LIN {X 0,Y 430.337,Z 1009.214,A -85,B 0,C 180,E1 10047.011,E2 10047.011} C_VEL
LIN {X 0,Y 422.721,Z 1027.569,A -85,B 0,C 180,E1 10045.411,E2 10045.411} C_VEL
LIN {X 0,Y 412.935,Z 1049.67,A -85,B 0,C 180,E1 10043.164,E2 10043.164} C_VEL
LIN {X 0,Y 403.725,Z 1069.015,A -85,B 0,C 180,E1 10040.822,E2 10040.822} C_VEL
LIN {X 0,Y 396.125,Z 1084.43,A -85,B 0,C 180,E1 10038.672,E2 10038.672} C_VEL
LIN {X 0,Y 389.035,Z 1098.425,A -85,B 0,C 180,E1 10036.451,E2 10036.451} C_VEL
LIN {X 0,Y 381.874,Z 1112.344,A -85,B 0,C 180,E1 10033.937,E2 10033.937} C_VEL
LIN {X 0,Y 373.58,Z 1128.48,A -85,B 0,C 180,E1 10030.571,E2 10030.571} C_VEL
LIN {X 0,Y 366.042,Z 1142.999,A -85,B 0,C 180,E1 10026.939,E2 10026.939} C_VEL
LIN {X 0,Y 360.784,Z 1153.631,A -85,B 0,C 180,E1 10023.853,E2 10023.853} C_VEL
LIN {X 0,Y 356.104,Z 1163.538,A -85,B 0,C 180,E1 10020.546,E2 10020.546} C_VEL
LIN {X 0,Y 351.983,Z 1173.044,A -85,B 0,C 180,E1 10016.851,E2 10016.851} C_VEL
LIN {X 0,Y 348.273,Z 1182.759,A -85,B 0,C 180,E1 10012.27,E2 10012.27} C_VEL
LIN {X 0,Y 346.233,Z 1189.194,A -85,B 0,C 180,E1 10008.522,E2 10008.522} C_VEL
LIN {X 0,Y 345,Z 1194.199,A -85,B 0,C 180,E1 10004.948,E2 10004.948} C_VEL
LIN {X 0,Y 344.316,Z 1197.956,A -85,B 0,C 180,E1 10001.559,E2 10001.559} C_VEL
LIN {X 0,Y 344.025,Z 1200.753,A -85,B 0,C 180,E1 9998.188,E2 9998.188} C_VEL
LIN {X 0,Y 343.928,Z 1202.539,A -85,B 0,C 180,E1 9995.004,E2 9995.004} C_VEL
LIN {X 0,Y 343.912,Z 1203.491,A -85,B 0,C 180,E1 9991.833,E2 9991.833} C_VEL
LIN {X 0,Y 343.916,Z 1203.616,A -85,B 0,C 180,E1 9988.668,E2 9988.668} C_VEL
LIN {X 0,Y 343.921,Z 1202.851,A -85,B 0,C 180,E1 9985.331,E2 9985.331} C_VEL
LIN {X 0,Y 344.027,Z 1201.059,A -85,B 0,C 180,E1 9981.813,E2 9981.813} C_VEL
LIN {X 0,Y 344.324,Z 1198.421,A -85,B 0,C 180,E1 9978.442,E2 9978.442} C_VEL
LIN {X 0,Y 345.068,Z 1194.647,A -85,B 0,C 180,E1 9974.884,E2 9974.884} C_VEL
LIN {X 0,Y 346.354,Z 1189.832,A -85,B 0,C 180,E1 9971.311,E2 9971.311} C_VEL
LIN {X 0,Y 348.358,Z 1183.946,A -85,B 0,C 180,E1 9967.737,E2 9967.737} C_VEL
LIN {X 0,Y 351.492,Z 1176.249,A -85,B 0,C 180,E1 9963.838,E2 9963.838} C_VEL
LIN {X 0,Y 356.789,Z 1164.942,A -85,B 0,C 180,E1 9959.147,E2 9959.147} C_VEL
LIN {X 0,Y 362.173,Z 1154.455,A -85,B 0,C 180,E1 9955.532,E2 9955.532} C_VEL
LIN {X 0,Y 368.045,Z 1143.651,A -85,B 0,C 180,E1 9952.32,E2 9952.32} C_VEL
LIN {X 0,Y 375.262,Z 1130.896,A -85,B 0,C 180,E1 9949.046,E2 9949.046} C_VEL
LIN {X 0,Y 385.141,Z 1113.513,A -85,B 0,C 180,E1 9945.288,E2 9945.288} C_VEL
LIN {X 0,Y 393.592,Z 1098.51,A -85,B 0,C 180,E1 9942.549,E2 9942.549} C_VEL
LIN {X 0,Y 401.844,Z 1083.635,A -85,B 0,C 180,E1 9940.193,E2 9940.193} C_VEL
LIN {X 0,Y 410.984,Z 1066.687,A -85,B 0,C 180,E1 9937.865,E2 9937.865} C_VEL
LIN {X 0,Y 422.46,Z 1044.207,A -85,B 0,C 180,E1 9935.261,E2 9935.261} C_VEL
LIN {X 0,Y 431.379,Z 1025.581,A -85,B 0,C 180,E1 9933.445,E2 9933.445} C_VEL
LIN {X 0,Y 439.453,Z 1007.671,A -85,B 0,C 180,E1 9931.933,E2 9931.933} C_VEL
LIN {X 0,Y 447.149,Z 989.316,A -85,B 0,C 180,E1 9930.583,E2 9930.583} C_VEL
LIN {X 0,Y 456.108,Z 966.119,A -85,B 0,C 180,E1 9929.122,E2 9929.122} C_VEL
LIN {X 0,Y 464.642,Z 940.864,A -85,B 0,C 180,E1 9927.818,E2 9927.818} C_VEL
LIN {X 0,Y 470.596,Z 921.068,A -85,B 0,C 180,E1 9926.963,E2 9926.963} C_VEL
LIN {X 0,Y 476.118,Z 900.238,A -85,B 0,C 180,E1 9926.202,E2 9926.202} C_VEL
LIN {X 0,Y 481.006,Z 878.867,A -85,B 0,C 180,E1 9925.557,E2 9925.557} C_VEL
LIN {X 0,Y 485.675,Z 854.323,A -85,B 0,C 180,E1 9924.964,E2 9924.964} C_VEL
LIN {X 0,Y 489.575,Z 825.773,A -85,B 0,C 180,E1 9924.432,E2 9924.432} C_VEL
LIN {X 0,Y 495.874,Z 750.481,A -85,B 0,C 180,E1 9923.248,E2 9923.248} C_VEL
LIN {X 0,Y 512.566,Z 549.481,A -85,B 0,C 180,E1 9920.146,E2 9920.146} C_VEL
LIN {X 0,Y 508.739,Z 542.747,A -85,B 0,C 180,E1 9918.388,E2 9918.388} C_VEL
LIN {X 0,Y 504.17,Z 535.587,A -85,B 0,C 180,E1 9916.002,E2 9916.002} C_VEL
LIN {X 0,Y 501.343,Z 531.216,A -85,B 0,C 180,E1 9914.259,E2 9914.259} C_VEL
LIN {X 0,Y 498.781,Z 527.221,A -85,B 0,C 180,E1 9912.386,E2 9912.386} C_VEL
LIN {X 0,Y 496.043,Z 522.871,A -85,B 0,C 180,E1 9909.807,E2 9909.807} C_VEL
LIN {X 0,Y 493.101,Z 516.967,A -85,B 0,C 180,E1 9903.022,E2 9903.022} C_VEL
LIN {X 0,Y 493.133,Z 517.942,A -85,B 0,C 180,E1 9901.51,E2 9901.51} C_VEL
LIN {X 0,Y 495.468,Z 522.125,A -85,B 0,C 180,E1 9896.645,E2 9896.645} C_VEL
LIN {X 0,Y 496.115,Z 523.083,A -85,B 0,C 180,E1 9895.897,E2 9895.897} C_VEL
LIN {X 0,Y 499.395,Z 528.172,A -85,B 0,C 180,E1 9892.927,E2 9892.927} C_VEL
LIN {X 0,Y 502.886,Z 533.499,A -85,B 0,C 180,E1 9890.559,E2 9890.559} C_VEL
LIN {X 0,Y 506.125,Z 538.595,A -85,B 0,C 180,E1 9888.721,E2 9888.721} C_VEL
LIN {X 0,Y 510.891,Z 546.035,A -85,B 0,C 180,E1 9886.417,E2 9886.417} C_VEL
LIN {X 0,Y 512.516,Z 548.924,A -85,B 0,C 180,E1 9885.693,E2 9885.693} C_VEL
LIN {X 0,Y 495.201,Z 757.347,A -85,B 0,C 180,E1 9882.478,E2 9882.478} C_VEL
LIN {X 0,Y 489.709,Z 822.286,A -85,B 0,C 180,E1 9881.456,E2 9881.456} C_VEL
LIN {X 0,Y 485.517,Z 852.232,A -85,B 0,C 180,E1 9880.882,E2 9880.882} C_VEL
LIN {X 0,Y 481.117,Z 875.351,A -85,B 0,C 180,E1 9880.303,E2 9880.303} C_VEL
LIN {X 0,Y 476.393,Z 896.103,A -85,B 0,C 180,E1 9879.66,E2 9879.66} C_VEL
LIN {X 0,Y 471.007,Z 916.496,A -85,B 0,C 180,E1 9878.904,E2 9878.904} C_VEL
LIN {X 0,Y 464.448,Z 938.347,A -85,B 0,C 180,E1 9877.939,E2 9877.939} C_VEL
LIN {X 0,Y 455.544,Z 964.201,A -85,B 0,C 180,E1 9876.558,E2 9876.558} C_VEL
LIN {X 0,Y 447.584,Z 984.742,A -85,B 0,C 180,E1 9875.242,E2 9875.242} C_VEL
LIN {X 0,Y 439.887,Z 1003.084,A -85,B 0,C 180,E1 9873.875,E2 9873.875} C_VEL
LIN {X 0,Y 432.098,Z 1020.324,A -85,B 0,C 180,E1 9872.406,E2 9872.406} C_VEL
LIN {X 0,Y 423.37,Z 1038.473,A -85,B 0,C 180,E1 9870.628,E2 9870.628} C_VEL
LIN {X 0,Y 412.195,Z 1060.31,A -85,B 0,C 180,E1 9868.102,E2 9868.102} C_VEL
LIN {X 0,Y 402.856,Z 1077.491,A -85,B 0,C 180,E1 9865.739,E2 9865.739} C_VEL
LIN {X 0,Y 394.672,Z 1092.083,A -85,B 0,C 180,E1 9863.426,E2 9863.426} C_VEL
LIN {X 0,Y 386.658,Z 1106.09,A -85,B 0,C 180,E1 9860.875,E2 9860.875} C_VEL
LIN {X 0,Y 377.588,Z 1121.928,A -85,B 0,C 180,E1 9857.525,E2 9857.525} C_VEL
LIN {X 0,Y 369.258,Z 1136.254,A -85,B 0,C 180,E1 9853.883,E2 9853.883} C_VEL
LIN {X 0,Y 363.271,Z 1146.929,A -85,B 0,C 180,E1 9850.716,E2 9850.716} C_VEL
LIN {X 0,Y 358.211,Z 1156.378,A -85,B 0,C 180,E1 9847.481,E2 9847.481} C_VEL
LIN {X 0,Y 353.653,Z 1165.506,A -85,B 0,C 180,E1 9843.846,E2 9843.846} C_VEL
LIN {X 0,Y 349.353,Z 1175.205,A -85,B 0,C 180,E1 9839.196,E2 9839.196} C_VEL
LIN {X 0,Y 346.772,Z 1182.05,A -85,B 0,C 180,E1 9835.078,E2 9835.078} C_VEL
LIN {X 0,Y 345.352,Z 1186.792,A -85,B 0,C 180,E1 9831.573,E2 9831.573} C_VEL
LIN {X 0,Y 344.516,Z 1190.531,A -85,B 0,C 180,E1 9828.091,E2 9828.091} C_VEL
LIN {X 0,Y 344.106,Z 1193.313,A -85,B 0,C 180,E1 9824.619,E2 9824.619} C_VEL
LIN {X 0,Y 343.953,Z 1195.053,A -85,B 0,C 180,E1 9821.4,E2 9821.4} C_VEL
LIN {X 0,Y 343.924,Z 1195.977,A -85,B 0,C 180,E1 9818.189,E2 9818.189} C_VEL
LIN {X 0,Y 343.906,Z 1196.085,A -85,B 0,C 180,E1 9815.003,E2 9815.003} C_VEL
LIN {X 0,Y 343.931,Z 1195.318,A -85,B 0,C 180,E1 9811.665,E2 9811.665} C_VEL
LIN {X 0,Y 344.029,Z 1193.662,A -85,B 0,C 180,E1 9808.334,E2 9808.334} C_VEL
LIN {X 0,Y 344.331,Z 1190.956,A -85,B 0,C 180,E1 9804.835,E2 9804.835} C_VEL
LIN {X 0,Y 345.031,Z 1187.255,A -85,B 0,C 180,E1 9801.332,E2 9801.332} C_VEL
LIN {X 0,Y 346.236,Z 1182.539,A -85,B 0,C 180,E1 9797.829,E2 9797.829} C_VEL
LIN {X 0,Y 348.088,Z 1176.778,A -85,B 0,C 180,E1 9794.334,E2 9794.334} C_VEL
LIN {X 0,Y 350.975,Z 1169.245,A -85,B 0,C 180,E1 9790.529,E2 9790.529} C_VEL
LIN {X 0,Y 355.826,Z 1158.156,A -85,B 0,C 180,E1 9785.955,E2 9785.955} C_VEL
LIN {X 0,Y 360.768,Z 1147.87,A -85,B 0,C 180,E1 9782.429,E2 9782.429} C_VEL
LIN {X 0,Y 366.116,Z 1137.271,A -85,B 0,C 180,E1 9779.289,E2 9779.289} C_VEL
LIN {X 0,Y 372.644,Z 1124.746,A -85,B 0,C 180,E1 9776.075,E2 9776.075} C_VEL
LIN {X 0,Y 375.605,Z 1119.162,A -85,B 0,C 180,E1 9774.794,E2 9774.794} C_VEL
LIN {X 0,Y 376.92,Z 1115.143,A -85,B 0,C 180,E1 9773.809,E2 9773.809} C_VEL
LIN {X 0,Y 377.577,Z 1105.226,A -85,B 0,C 180,E1 9771.149,E2 9771.149} C_VEL
LIN {X 0,Y 379.228,Z 1100.831,A -85,B 0,C 180,E1 9770.204,E2 9770.204} C_VEL
LIN {X 0,Y 389.048,Z 1082.432,A -85,B 0,C 180,E1 9767.072,E2 9767.072} C_VEL
LIN {X 0,Y 397.703,Z 1065.618,A -85,B 0,C 180,E1 9764.642,E2 9764.642} C_VEL
LIN {X 0,Y 405.643,Z 1049.578,A -85,B 0,C 180,E1 9762.626,E2 9762.626} C_VEL
LIN {X 0,Y 414.307,Z 1031.223,A -85,B 0,C 180,E1 9760.623,E2 9760.623} C_VEL
LIN {X 0,Y 424.867,Z 1007.083,A -85,B 0,C 180,E1 9758.401,E2 9758.401} C_VEL
LIN {X 0,Y 432.771,Z 987.358,A -85,B 0,C 180,E1 9756.87,E2 9756.87} C_VEL
LIN {X 0,Y 440.027,Z 967.758,A -85,B 0,C 180,E1 9755.562,E2 9755.562} C_VEL
LIN {X 0,Y 446.974,Z 947.041,A -85,B 0,C 180,E1 9754.365,E2 9754.365} C_VEL
LIN {X 0,Y 455.108,Z 919.496,A -85,B 0,C 180,E1 9753.053,E2 9753.053} C_VEL
LIN {X 0,Y 460.585,Z 897.814,A -85,B 0,C 180,E1 9752.209,E2 9752.209} C_VEL
LIN {X 0,Y 465.192,Z 876.616,A -85,B 0,C 180,E1 9751.522,E2 9751.522} C_VEL
LIN {X 0,Y 469.15,Z 854.894,A -85,B 0,C 180,E1 9750.948,E2 9750.948} C_VEL
LIN {X 0,Y 473.042,Z 827.866,A -85,B 0,C 180,E1 9750.39,E2 9750.39} C_VEL
LIN {X 0,Y 476.588,Z 784.854,A -85,B 0,C 180,E1 9749.693,E2 9749.693} C_VEL
LIN {X 0,Y 493.006,Z 566.419,A -85,B 0,C 180,E1 9746.295,E2 9746.295} C_VEL
LIN {X 0,Y 494.586,Z 545.42,A -85,B 0,C 180,E1 9745.957,E2 9745.957} C_VEL
LIN {X 0,Y 487.433,Z 533.892,A -85,B 0,C 180,E1 9743.355,E2 9743.355} C_VEL
LIN {X 0,Y 480.969,Z 523.893,A -85,B 0,C 180,E1 9740.633,E2 9740.633} C_VEL
LIN {X 0,Y 475.999,Z 516.443,A -85,B 0,C 180,E1 9738.176,E2 9738.176} C_VEL
LIN {X 0,Y 472.598,Z 511.532,A -85,B 0,C 180,E1 9736.217,E2 9736.217} C_VEL
LIN {X 0,Y 469.595,Z 507.098,A -85,B 0,C 180,E1 9734.174,E2 9734.174} C_VEL
LIN {X 0,Y 466.586,Z 502.594,A -85,B 0,C 180,E1 9731.621,E2 9731.621} C_VEL
LIN {X 0,Y 463.469,Z 498.329,A -85,B 0,C 180,E1 9727.687,E2 9727.687} C_VEL
LIN {X 0,Y 462.965,Z 496.787,A -85,B 0,C 180,E1 9726.448,E2 9726.448} C_VEL
LIN {X 0,Y 462.675,Z 496.688,A -85,B 0,C 180,E1 9720.371,E2 9720.371} C_VEL
LIN {X 0,Y 463.125,Z 497.115,A -85,B 0,C 180,E1 9719.258,E2 9719.258} C_VEL
LIN {X 0,Y 464.849,Z 500.839,A -85,B 0,C 180,E1 9716.3,E2 9716.3} C_VEL
LIN {X 0,Y 466.718,Z 502.888,A -85,B 0,C 180,E1 9714.344,E2 9714.344} C_VEL
LIN {X 0,Y 469.77,Z 507.346,A -85,B 0,C 180,E1 9711.801,E2 9711.801} C_VEL
LIN {X 0,Y 473.776,Z 513.252,A -85,B 0,C 180,E1 9709.174,E2 9709.174} C_VEL
LIN {X 0,Y 478.001,Z 519.572,A -85,B 0,C 180,E1 9706.882,E2 9706.882} C_VEL
LIN {X 0,Y 482.852,Z 526.838,A -85,B 0,C 180,E1 9704.629,E2 9704.629} C_VEL
LIN {X 0,Y 489.094,Z 536.563,A -85,B 0,C 180,E1 9702.111,E2 9702.111} C_VEL
LIN {X 0,Y 493.408,Z 544.162,A -85,B 0,C 180,E1 9700.527,E2 9700.527} C_VEL
LIN {X 0,Y 494.638,Z 546.737,A -85,B 0,C 180,E1 9700.084,E2 9700.084} C_VEL
LIN {X 0,Y 477.921,Z 768.344,A -85,B 0,C 180,E1 9696.639,E2 9696.639} C_VEL
LIN {X 0,Y 473.332,Z 827.257,A -85,B 0,C 180,E1 9695.7,E2 9695.7} C_VEL
LIN {X 0,Y 469.295,Z 857.376,A -85,B 0,C 180,E1 9695.108,E2 9695.108} C_VEL
LIN {X 0,Y 465.131,Z 880.202,A -85,B 0,C 180,E1 9694.528,E2 9694.528} C_VEL
LIN {X 0,Y 460.653,Z 900.854,A -85,B 0,C 180,E1 9693.878,E2 9693.878} C_VEL
LIN {X 0,Y 455.634,Z 920.879,A -85,B 0,C 180,E1 9693.123,E2 9693.123} C_VEL
LIN {X 0,Y 449.408,Z 942.77,A -85,B 0,C 180,E1 9692.145,E2 9692.145} C_VEL
LIN {X 0,Y 440.755,Z 969.366,A -85,B 0,C 180,E1 9690.702,E2 9690.702} C_VEL
LIN {X 0,Y 433.36,Z 989.619,A -85,B 0,C 180,E1 9689.386,E2 9689.386} C_VEL
LIN {X 0,Y 425.854,Z 1008.604,A -85,B 0,C 180,E1 9687.953,E2 9687.953} C_VEL
LIN {X 0,Y 418.291,Z 1026.382,A -85,B 0,C 180,E1 9686.414,E2 9686.414} C_VEL
LIN {X 0,Y 409.052,Z 1046.833,A -85,B 0,C 180,E1 9684.367,E2 9684.367} C_VEL
LIN {X 0,Y 398.982,Z 1067.537,A -85,B 0,C 180,E1 9681.898,E2 9681.898} C_VEL
LIN {X 0,Y 390.791,Z 1083.647,A -85,B 0,C 180,E1 9679.659,E2 9679.659} C_VEL
LIN {X 0,Y 383.252,Z 1098.048,A -85,B 0,C 180,E1 9677.368,E2 9677.368} C_VEL
LIN {X 0,Y 375.365,Z 1112.862,A -85,B 0,C 180,E1 9674.665,E2 9674.665} C_VEL
LIN {X 0,Y 366.459,Z 1129.485,A -85,B 0,C 180,E1 9671.115,E2 9671.115} C_VEL
LIN {X 0,Y 359.007,Z 1143.306,A -85,B 0,C 180,E1 9667.586,E2 9667.586} C_VEL
LIN {X 0,Y 353.534,Z 1153.902,A -85,B 0,C 180,E1 9664.448,E2 9664.448} C_VEL
LIN {X 0,Y 348.669,Z 1163.773,A -85,B 0,C 180,E1 9661.077,E2 9661.077} C_VEL
LIN {X 0,Y 343.854,Z 1174.5,A -85,B 0,C 180,E1 9656.782,E2 9656.782} C_VEL
LIN {X 0,Y 340.36,Z 1183.199,A -85,B 0,C 180,E1 9652.452,E2 9652.452} C_VEL
LIN {X 0,Y 338.336,Z 1189.291,A -85,B 0,C 180,E1 9648.792,E2 9648.792} C_VEL
LIN {X 0,Y 337.091,Z 1194.053,A -85,B 0,C 180,E1 9645.308,E2 9645.308} C_VEL
LIN {X 0,Y 336.353,Z 1197.825,A -85,B 0,C 180,E1 9641.837,E2 9641.837} C_VEL
LIN {X 0,Y 336.036,Z 1200.635,A -85,B 0,C 180,E1 9638.384,E2 9638.384} C_VEL
LIN {X 0,Y 335.93,Z 1202.433,A -85,B 0,C 180,E1 9635.124,E2 9635.124} C_VEL
LIN {X 0,Y 335.913,Z 1203.397,A -85,B 0,C 180,E1 9631.877,E2 9631.877} C_VEL
LIN {X 0,Y 335.916,Z 1203.535,A -85,B 0,C 180,E1 9628.636,E2 9628.636} C_VEL
LIN {X 0,Y 335.923,Z 1202.781,A -85,B 0,C 180,E1 9625.22,E2 9625.22} C_VEL
LIN {X 0,Y 336.036,Z 1201,A -85,B 0,C 180,E1 9621.617,E2 9621.617} C_VEL
LIN {X 0,Y 336.361,Z 1198.374,A -85,B 0,C 180,E1 9618.165,E2 9618.165} C_VEL
LIN {X 0,Y 337.166,Z 1194.615,A -85,B 0,C 180,E1 9614.521,E2 9614.521} C_VEL
LIN {X 0,Y 338.547,Z 1189.813,A -85,B 0,C 180,E1 9610.864,E2 9610.864} C_VEL
LIN {X 0,Y 340.694,Z 1183.943,A -85,B 0,C 180,E1 9607.208,E2 9607.208} C_VEL
LIN {X 0,Y 343.855,Z 1176.617,A -85,B 0,C 180,E1 9603.398,E2 9603.398} C_VEL
LIN {X 0,Y 349.172,Z 1165.906,A -85,B 0,C 180,E1 9598.782,E2 9598.782} C_VEL
LIN {X 0,Y 355.003,Z 1155.038,A -85,B 0,C 180,E1 9594.931,E2 9594.931} C_VEL
LIN {X 0,Y 361.115,Z 1144.315,A -85,B 0,C 180,E1 9591.668,E2 9591.668} C_VEL
LIN {X 0,Y 368.027,Z 1132.577,A -85,B 0,C 180,E1 9588.579,E2 9588.579} C_VEL
LIN {X 0,Y 377.097,Z 1117.416,A -85,B 0,C 180,E1 9585.147,E2 9585.147} C_VEL
LIN {X 0,Y 387.052,Z 1100.377,A -85,B 0,C 180,E1 9581.928,E2 9581.928} C_VEL
LIN {X 0,Y 396.019,Z 1084.777,A -85,B 0,C 180,E1 9579.414,E2 9579.414} C_VEL
LIN {X 0,Y 404.635,Z 1069.353,A -85,B 0,C 180,E1 9577.259,E2 9577.259} C_VEL
LIN {X 0,Y 413.667,Z 1052.517,A -85,B 0,C 180,E1 9575.218,E2 9575.218} C_VEL
LIN {X 0,Y 424.884,Z 1030.346,A -85,B 0,C 180,E1 9572.93,E2 9572.93} C_VEL
LIN {X 0,Y 434.172,Z 1010.429,A -85,B 0,C 180,E1 9571.21,E2 9571.21} C_VEL
LIN {X 0,Y 442.148,Z 992.041,A -85,B 0,C 180,E1 9569.836,E2 9569.836} C_VEL
LIN {X 0,Y 449.827,Z 972.877,A -85,B 0,C 180,E1 9568.599,E2 9568.599} C_VEL
LIN {X 0,Y 457.246,Z 952.607,A -85,B 0,C 180,E1 9567.478,E2 9567.478} C_VEL
LIN {X 0,Y 465.609,Z 926.935,A -85,B 0,C 180,E1 9566.291,E2 9566.291} C_VEL
LIN {X 0,Y 472.3,Z 902.65,A -85,B 0,C 180,E1 9565.387,E2 9565.387} C_VEL
LIN {X 0,Y 477.432,Z 880.973,A -85,B 0,C 180,E1 9564.726,E2 9564.726} C_VEL
LIN {X 0,Y 481.653,Z 859.76,A -85,B 0,C 180,E1 9564.203,E2 9564.203} C_VEL
LIN {X 0,Y 485.58,Z 834.829,A -85,B 0,C 180,E1 9563.709,E2 9563.709} C_VEL
LIN {X 0,Y 489.174,Z 798.01,A -85,B 0,C 180,E1 9563.109,E2 9563.109} C_VEL
LIN {X 0,Y 507.912,Z 575.83,A -85,B 0,C 180,E1 9559.692,E2 9559.692} C_VEL
LIN {X 0,Y 509.714,Z 554.831,A -85,B 0,C 180,E1 9559.361,E2 9559.361} C_VEL
LIN {X 0,Y 505.974,Z 548.265,A -85,B 0,C 180,E1 9557.54,E2 9557.54} C_VEL
LIN {X 0,Y 502.226,Z 542.441,A -85,B 0,C 180,E1 9555.473,E2 9555.473} C_VEL
LIN {X 0,Y 499.942,Z 538.803,A -85,B 0,C 180,E1 9554.005,E2 9554.005} C_VEL
LIN {X 0,Y 497.519,Z 534.955,A -85,B 0,C 180,E1 9552.182,E2 9552.182} C_VEL
LIN {X 0,Y 494.879,Z 530.602,A -85,B 0,C 180,E1 9549.61,E2 9549.61} C_VEL
LIN {X 0,Y 492.117,Z 525.419,A -85,B 0,C 180,E1 9543.728,E2 9543.728} C_VEL
LIN {X 0,Y 492.128,Z 524.917,A -85,B 0,C 180,E1 9542.678,E2 9542.678} C_VEL
LIN {X 0,Y 494.389,Z 530.008,A -85,B 0,C 180,E1 9536.754,E2 9536.754} C_VEL
LIN {X 0,Y 495.021,Z 530.988,A -85,B 0,C 180,E1 9536.004,E2 9536.004} C_VEL
LIN {X 0,Y 498.178,Z 535.986,A -85,B 0,C 180,E1 9533.083,E2 9533.083} C_VEL
LIN {X 0,Y 501.521,Z 541.18,A -85,B 0,C 180,E1 9530.764,E2 9530.764} C_VEL
LIN {X 0,Y 504.699,Z 546.29,A -85,B 0,C 180,E1 9528.92,E2 9528.92} C_VEL
LIN {X 0,Y 509.327,Z 553.688,A -85,B 0,C 180,E1 9526.634,E2 9526.634} C_VEL
LIN {X 0,Y 509.654,Z 554.618,A -85,B 0,C 180,E1 9526.467,E2 9526.467} C_VEL
LIN {X 0,Y 491.699,Z 765.89,A -85,B 0,C 180,E1 9523.22,E2 9523.22} C_VEL
LIN {X 0,Y 486.687,Z 823.199,A -85,B 0,C 180,E1 9522.319,E2 9522.319} C_VEL
LIN {X 0,Y 482.354,Z 853.133,A -85,B 0,C 180,E1 9521.745,E2 9521.745} C_VEL
LIN {X 0,Y 477.962,Z 875.7,A -85,B 0,C 180,E1 9521.184,E2 9521.184} C_VEL
LIN {X 0,Y 473.183,Z 896.258,A -85,B 0,C 180,E1 9520.553,E2 9520.553} C_VEL
LIN {X 0,Y 467.503,Z 917.296,A -85,B 0,C 180,E1 9519.779,E2 9519.779} C_VEL
LIN {X 0,Y 459.94,Z 941.852,A -85,B 0,C 180,E1 9518.69,E2 9518.69} C_VEL
LIN {X 0,Y 451.18,Z 966.167,A -85,B 0,C 180,E1 9517.37,E2 9517.37} C_VEL
LIN {X 0,Y 443.411,Z 985.678,A -85,B 0,C 180,E1 9516.117,E2 9516.117} C_VEL
LIN {X 0,Y 435.536,Z 1003.933,A -85,B 0,C 180,E1 9514.757,E2 9514.757} C_VEL
LIN {X 0,Y 427.233,Z 1021.787,A -85,B 0,C 180,E1 9513.231,E2 9513.231} C_VEL
LIN {X 0,Y 416.762,Z 1042.929,A -85,B 0,C 180,E1 9511.125,E2 9511.125} C_VEL
LIN {X 0,Y 405.951,Z 1062.989,A -85,B 0,C 180,E1 9508.723,E2 9508.723} C_VEL
LIN {X 0,Y 397.16,Z 1078.624,A -85,B 0,C 180,E1 9506.54,E2 9506.54} C_VEL
LIN {X 0,Y 388.54,Z 1093.452,A -85,B 0,C 180,E1 9504.156,E2 9504.156} C_VEL
LIN {X 0,Y 378.838,Z 1109.866,A -85,B 0,C 180,E1 9501.085,E2 9501.085} C_VEL
LIN {X 0,Y 369.067,Z 1125.951,A -85,B 0,C 180,E1 9497.467,E2 9497.467} C_VEL
LIN {X 0,Y 361.894,Z 1137.891,A -85,B 0,C 180,E1 9494.307,E2 9494.307} C_VEL
LIN {X 0,Y 355.798,Z 1148.309,A -85,B 0,C 180,E1 9491.116,E2 9491.116} C_VEL
LIN {X 0,Y 349.609,Z 1159.485,A -85,B 0,C 180,E1 9487.117,E2 9487.117} C_VEL
LIN {X 0,Y 344.198,Z 1170,A -85,B 0,C 180,E1 9482.507,E2 9482.507} C_VEL
LIN {X 0,Y 340.989,Z 1177.103,A -85,B 0,C 180,E1 9478.743,E2 9478.743} C_VEL
LIN {X 0,Y 338.743,Z 1182.956,A -85,B 0,C 180,E1 9475.015,E2 9475.015} C_VEL
LIN {X 0,Y 337.243,Z 1187.805,A -85,B 0,C 180,E1 9471.205,E2 9471.205} C_VEL
LIN {X 0,Y 336.353,Z 1191.972,A -85,B 0,C 180,E1 9466.937,E2 9466.937} C_VEL
LIN {X 0,Y 335.99,Z 1194.765,A -85,B 0,C 180,E1 9462.546,E2 9462.546} C_VEL
LIN {X 0,Y 335.925,Z 1196.009,A -85,B 0,C 180,E1 9458.731,E2 9458.731} C_VEL
LIN {X 0,Y 335.906,Z 1196.186,A -85,B 0,C 180,E1 9455.123,E2 9455.123} C_VEL
LIN {X 0,Y 335.931,Z 1195.444,A -85,B 0,C 180,E1 9451.705,E2 9451.705} C_VEL
LIN {X 0,Y 336.032,Z 1193.813,A -85,B 0,C 180,E1 9448.294,E2 9448.294} C_VEL
LIN {X 0,Y 336.348,Z 1191.134,A -85,B 0,C 180,E1 9444.712,E2 9444.712} C_VEL
LIN {X 0,Y 337.085,Z 1187.459,A -85,B 0,C 180,E1 9441.126,E2 9441.126} C_VEL
LIN {X 0,Y 338.363,Z 1182.768,A -85,B 0,C 180,E1 9437.542,E2 9437.542} C_VEL
LIN {X 0,Y 340.299,Z 1177.034,A -85,B 0,C 180,E1 9433.966,E2 9433.966} C_VEL
LIN {X 0,Y 343.03,Z 1170.217,A -85,B 0,C 180,E1 9430.414,E2 9430.414} C_VEL
LIN {X 0,Y 347.6,Z 1160.28,A -85,B 0,C 180,E1 9426.071,E2 9426.071} C_VEL
LIN {X 0,Y 353.312,Z 1148.738,A -85,B 0,C 180,E1 9421.979,E2 9421.979} C_VEL
LIN {X 0,Y 358.833,Z 1138.222,A -85,B 0,C 180,E1 9418.782,E2 9418.782} C_VEL
LIN {X 0,Y 365.224,Z 1126.409,A -85,B 0,C 180,E1 9415.669,E2 9415.669} C_VEL
LIN {X 0,Y 373.681,Z 1111.126,A -85,B 0,C 180,E1 9412.211,E2 9412.211} C_VEL
LIN {X 0,Y 379.228,Z 1100.831,A -85,B 0,C 180,E1 9410.204,E2 9410.204} C_VEL
LIN {X 0,Y 380.941,Z 1096.425,A -85,B 0,C 180,E1 9409.276,E2 9409.276} C_VEL
LIN {X 0,Y 382.709,Z 1084.847,A -85,B 0,C 180,E1 9406.621,E2 9406.621} C_VEL
LIN {X 0,Y 384.413,Z 1080.641,A -85,B 0,C 180,E1 9405.89,E2 9405.89} C_VEL
LIN {X 0,Y 392.59,Z 1065.226,A -85,B 0,C 180,E1 9403.671,E2 9403.671} C_VEL
LIN {X 0,Y 400.776,Z 1049.133,A -85,B 0,C 180,E1 9401.65,E2 9401.65} C_VEL
LIN {X 0,Y 410.276,Z 1029.531,A -85,B 0,C 180,E1 9399.525,E2 9399.525} C_VEL
LIN {X 0,Y 420.549,Z 1006.454,A -85,B 0,C 180,E1 9397.429,E2 9397.429} C_VEL
LIN {X 0,Y 428.491,Z 987.053,A -85,B 0,C 180,E1 9395.931,E2 9395.931} C_VEL
LIN {X 0,Y 435.765,Z 967.827,A -85,B 0,C 180,E1 9394.655,E2 9394.655} C_VEL
LIN {X 0,Y 442.874,Z 947.104,A -85,B 0,C 180,E1 9393.465,E2 9393.465} C_VEL
LIN {X 0,Y 451.182,Z 919.549,A -85,B 0,C 180,E1 9392.16,E2 9392.16} C_VEL
LIN {X 0,Y 456.775,Z 897.852,A -85,B 0,C 180,E1 9391.322,E2 9391.322} C_VEL
LIN {X 0,Y 461.468,Z 876.656,A -85,B 0,C 180,E1 9390.64,E2 9390.64} C_VEL
LIN {X 0,Y 465.531,Z 854.757,A -85,B 0,C 180,E1 9390.067,E2 9390.067} C_VEL
LIN {X 0,Y 469.524,Z 827.339,A -85,B 0,C 180,E1 9389.507,E2 9389.507} C_VEL
LIN {X 0,Y 473.257,Z 782.72,A -85,B 0,C 180,E1 9388.787,E2 9388.787} C_VEL
LIN {X 0,Y 490,Z 565.649,A -85,B 0,C 180,E1 9385.417,E2 9385.417} C_VEL
LIN {X 0,Y 491.118,Z 550.311,A -85,B 0,C 180,E1 9385.151,E2 9385.151} C_VEL
LIN {X 0,Y 483.282,Z 537.54,A -85,B 0,C 180,E1 9382.12,E2 9382.12} C_VEL
LIN {X 0,Y 477.417,Z 528.439,A -85,B 0,C 180,E1 9379.451,E2 9379.451} C_VEL
LIN {X 0,Y 473.721,Z 522.991,A -85,B 0,C 180,E1 9377.504,E2 9377.504} C_VEL
LIN {X 0,Y 471.049,Z 518.995,A -85,B 0,C 180,E1 9375.892,E2 9375.892} C_VEL
LIN {X 0,Y 468.295,Z 514.82,A -85,B 0,C 180,E1 9373.962,E2 9373.962} C_VEL
LIN {X 0,Y 464.997,Z 509.87,A -85,B 0,C 180,E1 9371.033,E2 9371.033} C_VEL
LIN {X 0,Y 462.549,Z 506.542,A -85,B 0,C 180,E1 9367.827,E2 9367.827} C_VEL
LIN {X 0,Y 461.939,Z 504.709,A -85,B 0,C 180,E1 9366.338,E2 9366.338} C_VEL
LIN {X 0,Y 461.697,Z 504.629,A -85,B 0,C 180,E1 9360.372,E2 9360.372} C_VEL
LIN {X 0,Y 462.089,Z 505.002,A -85,B 0,C 180,E1 9359.38,E2 9359.38} C_VEL
LIN {X 0,Y 463.767,Z 508.711,A -85,B 0,C 180,E1 9356.415,E2 9356.415} C_VEL
LIN {X 0,Y 465.54,Z 510.691,A -85,B 0,C 180,E1 9354.515,E2 9354.515} C_VEL
LIN {X 0,Y 468.449,Z 515.054,A -85,B 0,C 180,E1 9352.025,E2 9352.025} C_VEL
LIN {X 0,Y 472.376,Z 520.949,A -85,B 0,C 180,E1 9349.388,E2 9349.388} C_VEL
LIN {X 0,Y 476.532,Z 527.273,A -85,B 0,C 180,E1 9347.087,E2 9347.087} C_VEL
LIN {X 0,Y 481.308,Z 534.617,A -85,B 0,C 180,E1 9344.826,E2 9344.826} C_VEL
LIN {X 0,Y 487.109,Z 543.8,A -85,B 0,C 180,E1 9342.437,E2 9342.437} C_VEL
LIN {X 0,Y 491.238,Z 551.25,A -85,B 0,C 180,E1 9340.882,E2 9340.882} C_VEL
LIN {X 0,Y 474.641,Z 765.905,A -85,B 0,C 180,E1 9337.549,E2 9337.549} C_VEL
LIN {X 0,Y 469.793,Z 826.819,A -85,B 0,C 180,E1 9336.58,E2 9336.58} C_VEL
LIN {X 0,Y 465.656,Z 857.232,A -85,B 0,C 180,E1 9335.987,E2 9335.987} C_VEL
LIN {X 0,Y 461.432,Z 879.99,A -85,B 0,C 180,E1 9335.414,E2 9335.414} C_VEL
LIN {X 0,Y 456.877,Z 900.605,A -85,B 0,C 180,E1 9334.772,E2 9334.772} C_VEL
LIN {X 0,Y 451.588,Z 921.286,A -85,B 0,C 180,E1 9333.998,E2 9333.998} C_VEL
LIN {X 0,Y 445.032,Z 943.793,A -85,B 0,C 180,E1 9332.993,E2 9332.993} C_VEL
LIN {X 0,Y 436.471,Z 969.403,A -85,B 0,C 180,E1 9331.604,E2 9331.604} C_VEL
LIN {X 0,Y 428.808,Z 989.904,A -85,B 0,C 180,E1 9330.274,E2 9330.274} C_VEL
LIN {X 0,Y 421.487,Z 1007.993,A -85,B 0,C 180,E1 9328.914,E2 9328.914} C_VEL
LIN {X 0,Y 413.764,Z 1025.704,A -85,B 0,C 180,E1 9327.391,E2 9327.391} C_VEL
LIN {X 0,Y 404.779,Z 1045.064,A -85,B 0,C 180,E1 9325.468,E2 9325.468} C_VEL
LIN {X 0,Y 393.837,Z 1067.093,A -85,B 0,C 180,E1 9322.863,E2 9322.863} C_VEL
LIN {X 0,Y 385.172,Z 1083.608,A -85,B 0,C 180,E1 9320.56,E2 9320.56} C_VEL
LIN {X 0,Y 377.101,Z 1098.528,A -85,B 0,C 180,E1 9318.165,E2 9318.165} C_VEL
LIN {X 0,Y 368.898,Z 1113.415,A -85,B 0,C 180,E1 9315.411,E2 9315.411} C_VEL
LIN {X 0,Y 358.993,Z 1131.125,A -85,B 0,C 180,E1 9311.521,E2 9311.521} C_VEL
LIN {X 0,Y 352.023,Z 1143.613,A -85,B 0,C 180,E1 9308.259,E2 9308.259} C_VEL
LIN {X 0,Y 346.324,Z 1154.169,A -85,B 0,C 180,E1 9305.068,E2 9305.068} C_VEL
LIN {X 0,Y 340.99,Z 1164.562,A -85,B 0,C 180,E1 9301.427,E2 9301.427} C_VEL
LIN {X 0,Y 335.56,Z 1176.102,A -85,B 0,C 180,E1 9296.549,E2 9296.549} C_VEL
LIN {X 0,Y 332.45,Z 1183.636,A -85,B 0,C 180,E1 9292.643,E2 9292.643} C_VEL
LIN {X 0,Y 330.445,Z 1189.387,A -85,B 0,C 180,E1 9289.075,E2 9289.075} C_VEL
LIN {X 0,Y 329.14,Z 1194.115,A -85,B 0,C 180,E1 9285.506,E2 9285.506} C_VEL
LIN {X 0,Y 328.368,Z 1197.854,A -85,B 0,C 180,E1 9281.951,E2 9281.951} C_VEL
LIN {X 0,Y 328.047,Z 1200.516,A -85,B 0,C 180,E1 9278.59,E2 9278.59} C_VEL
LIN {X 0,Y 327.933,Z 1202.327,A -85,B 0,C 180,E1 9275.249,E2 9275.249} C_VEL
LIN {X 0,Y 327.913,Z 1203.304,A -85,B 0,C 180,E1 9271.923,E2 9271.923} C_VEL
LIN {X 0,Y 327.915,Z 1203.43,A -85,B 0,C 180,E1 9268.428,E2 9268.428} C_VEL
LIN {X 0,Y 327.928,Z 1202.642,A -85,B 0,C 180,E1 9264.928,E2 9264.928} C_VEL
LIN {X 0,Y 328.049,Z 1200.943,A -85,B 0,C 180,E1 9261.411,E2 9261.411} C_VEL
LIN {X 0,Y 328.437,Z 1198.169,A -85,B 0,C 180,E1 9257.696,E2 9257.696} C_VEL
LIN {X 0,Y 329.273,Z 1194.583,A -85,B 0,C 180,E1 9254.14,E2 9254.14} C_VEL
LIN {X 0,Y 330.76,Z 1189.797,A -85,B 0,C 180,E1 9250.395,E2 9250.395} C_VEL
LIN {X 0,Y 333.057,Z 1183.943,A -85,B 0,C 180,E1 9246.655,E2 9246.655} C_VEL
LIN {X 0,Y 336.496,Z 1176.475,A -85,B 0,C 180,E1 9242.682,E2 9242.682} C_VEL
LIN {X 0,Y 342.283,Z 1165.503,A -85,B 0,C 180,E1 9237.883,E2 9237.883} C_VEL
LIN {X 0,Y 348.467,Z 1154.603,A -85,B 0,C 180,E1 9233.97,E2 9233.97} C_VEL
LIN {X 0,Y 354.936,Z 1143.842,A -85,B 0,C 180,E1 9230.667,E2 9230.667} C_VEL
LIN {X 0,Y 362.429,Z 1131.671,A -85,B 0,C 180,E1 9227.444,E2 9227.444} C_VEL
LIN {X 0,Y 372.547,Z 1115.378,A -85,B 0,C 180,E1 9223.784,E2 9223.784} C_VEL
LIN {X 0,Y 382.524,Z 1098.907,A -85,B 0,C 180,E1 9220.71,E2 9220.71} C_VEL
LIN {X 0,Y 391.336,Z 1084.094,A -85,B 0,C 180,E1 9218.336,E2 9218.336} C_VEL
LIN {X 0,Y 400.764,Z 1067.711,A -85,B 0,C 180,E1 9216.066,E2 9216.066} C_VEL
LIN {X 0,Y 411.994,Z 1047.279,A -85,B 0,C 180,E1 9213.652,E2 9213.652} C_VEL
LIN {X 0,Y 422.594,Z 1026.342,A -85,B 0,C 180,E1 9211.596,E2 9211.596} C_VEL
LIN {X 0,Y 431.385,Z 1007.84,A -85,B 0,C 180,E1 9210.044,E2 9210.044} C_VEL
LIN {X 0,Y 439.143,Z 990.287,A -85,B 0,C 180,E1 9208.767,E2 9208.767} C_VEL
LIN {X 0,Y 447.078,Z 970.771,A -85,B 0,C 180,E1 9207.533,E2 9207.533} C_VEL
LIN {X 0,Y 455.966,Z 946.725,A -85,B 0,C 180,E1 9206.25,E2 9206.25} C_VEL
LIN {X 0,Y 463.951,Z 921.458,A -85,B 0,C 180,E1 9205.157,E2 9205.157} C_VEL
LIN {X 0,Y 469.693,Z 900.717,A -85,B 0,C 180,E1 9204.415,E2 9204.415} C_VEL
LIN {X 0,Y 474.719,Z 879.675,A -85,B 0,C 180,E1 9203.791,E2 9203.791} C_VEL
LIN {X 0,Y 479.155,Z 857.476,A -85,B 0,C 180,E1 9203.258,E2 9203.258} C_VEL
LIN {X 0,Y 483.554,Z 828.156,A -85,B 0,C 180,E1 9202.705,E2 9202.705} C_VEL
LIN {X 0,Y 488.217,Z 776.531,A -85,B 0,C 180,E1 9201.893,E2 9201.893} C_VEL
LIN {X 0,Y 506.997,Z 560.235,A -85,B 0,C 180,E1 9198.584,E2 9198.584} C_VEL
LIN {X 0,Y 503.189,Z 553.892,A -85,B 0,C 180,E1 9196.627,E2 9196.627} C_VEL
LIN {X 0,Y 499.235,Z 547.297,A -85,B 0,C 180,E1 9194.208,E2 9194.208} C_VEL
LIN {X 0,Y 496.264,Z 542.688,A -85,B 0,C 180,E1 9191.978,E2 9191.978} C_VEL
LIN {X 0,Y 493.446,Z 538.034,A -85,B 0,C 180,E1 9189.094,E2 9189.094} C_VEL
LIN {X 0,Y 491.139,Z 533.73,A -85,B 0,C 180,E1 9184.014,E2 9184.014} C_VEL
LIN {X 0,Y 491.149,Z 532.845,A -85,B 0,C 180,E1 9182.801,E2 9182.801} C_VEL
LIN {X 0,Y 493.511,Z 538.047,A -85,B 0,C 180,E1 9176.632,E2 9176.632} C_VEL
LIN {X 0,Y 496.964,Z 543.797,A -85,B 0,C 180,E1 9173.24,E2 9173.24} C_VEL
LIN {X 0,Y 500.162,Z 548.861,A -85,B 0,C 180,E1 9170.971,E2 9170.971} C_VEL
LIN {X 0,Y 503.485,Z 554.313,A -85,B 0,C 180,E1 9169.009,E2 9169.009} C_VEL
LIN {X 0,Y 506.919,Z 559.981,A -85,B 0,C 180,E1 9167.255,E2 9167.255} C_VEL
LIN {X 0,Y 488.401,Z 773.039,A -85,B 0,C 180,E1 9163.994,E2 9163.994} C_VEL
LIN {X 0,Y 483.742,Z 824.452,A -85,B 0,C 180,E1 9163.187,E2 9163.187} C_VEL
LIN {X 0,Y 479.386,Z 853.582,A -85,B 0,C 180,E1 9162.63,E2 9162.63} C_VEL
LIN {X 0,Y 474.949,Z 875.938,A -85,B 0,C 180,E1 9162.08,E2 9162.08} C_VEL
LIN {X 0,Y 470.091,Z 896.432,A -85,B 0,C 180,E1 9161.458,E2 9161.458} C_VEL
LIN {X 0,Y 464.495,Z 916.791,A -85,B 0,C 180,E1 9160.718,E2 9160.718} C_VEL
LIN {X 0,Y 457.663,Z 938.61,A -85,B 0,C 180,E1 9159.774,E2 9159.774} C_VEL
LIN {X 0,Y 448.007,Z 965.358,A -85,B 0,C 180,E1 9158.364,E2 9158.364} C_VEL
LIN {X 0,Y 439.702,Z 985.79,A -85,B 0,C 180,E1 9157.066,E2 9157.066} C_VEL
LIN {X 0,Y 431.981,Z 1003.281,A -85,B 0,C 180,E1 9155.776,E2 9155.776} C_VEL
LIN {X 0,Y 423.784,Z 1020.506,A -85,B 0,C 180,E1 9154.327,E2 9154.327} C_VEL
LIN {X 0,Y 414.264,Z 1039.269,A -85,B 0,C 180,E1 9152.498,E2 9152.498} C_VEL
LIN {X 0,Y 402.136,Z 1061.509,A -85,B 0,C 180,E1 9149.912,E2 9149.912} C_VEL
LIN {X 0,Y 392.511,Z 1078.116,A -85,B 0,C 180,E1 9147.612,E2 9147.612} C_VEL
LIN {X 0,Y 383.512,Z 1093.093,A -85,B 0,C 180,E1 9145.209,E2 9145.209} C_VEL
LIN {X 0,Y 374.457,Z 1107.808,A -85,B 0,C 180,E1 9142.47,E2 9142.47} C_VEL
LIN {X 0,Y 363.657,Z 1125.048,A -85,B 0,C 180,E1 9138.642,E2 9138.642} C_VEL
LIN {X 0,Y 355.774,Z 1137.562,A -85,B 0,C 180,E1 9135.318,E2 9135.318} C_VEL
LIN {X 0,Y 349.273,Z 1148.116,A -85,B 0,C 180,E1 9132.057,E2 9132.057} C_VEL
LIN {X 0,Y 343.234,Z 1158.384,A -85,B 0,C 180,E1 9128.351,E2 9128.351} C_VEL
LIN {X 0,Y 337.135,Z 1169.534,A -85,B 0,C 180,E1 9123.479,E2 9123.479} C_VEL
LIN {X 0,Y 333.496,Z 1177.023,A -85,B 0,C 180,E1 9119.451,E2 9119.451} C_VEL
LIN {X 0,Y 331.116,Z 1182.713,A -85,B 0,C 180,E1 9115.774,E2 9115.774} C_VEL
LIN {X 0,Y 329.535,Z 1187.362,A -85,B 0,C 180,E1 9112.1,E2 9112.1} C_VEL
LIN {X 0,Y 328.591,Z 1191.01,A -85,B 0,C 180,E1 9108.448,E2 9108.448} C_VEL
LIN {X 0,Y 328.13,Z 1193.688,A -85,B 0,C 180,E1 9104.83,E2 9104.83} C_VEL
LIN {X 0,Y 327.952,Z 1195.424,A -85,B 0,C 180,E1 9101.251,E2 9101.251} C_VEL
LIN {X 0,Y 327.921,Z 1196.217,A -85,B 0,C 180,E1 9097.886,E2 9097.886} C_VEL
LIN {X 0,Y 327.911,Z 1196.195,A -85,B 0,C 180,E1 9094.546,E2 9094.546} C_VEL
LIN {X 0,Y 327.937,Z 1195.367,A -85,B 0,C 180,E1 9091.222,E2 9091.222} C_VEL
LIN {X 0,Y 328.052,Z 1193.74,A -85,B 0,C 180,E1 9087.903,E2 9087.903} C_VEL
LIN {X 0,Y 328.392,Z 1191.152,A -85,B 0,C 180,E1 9084.408,E2 9084.408} C_VEL
LIN {X 0,Y 329.16,Z 1187.583,A -85,B 0,C 180,E1 9080.844,E2 9080.844} C_VEL
LIN {X 0,Y 330.492,Z 1182.996,A -85,B 0,C 180,E1 9077.24,E2 9077.24} C_VEL
LIN {X 0,Y 332.524,Z 1177.288,A -85,B 0,C 180,E1 9073.581,E2 9073.581} C_VEL
LIN {X 0,Y 335.471,Z 1170.326,A -85,B 0,C 180,E1 9069.865,E2 9069.865} C_VEL
LIN {X 0,Y 340.176,Z 1160.595,A -85,B 0,C 180,E1 9065.515,E2 9065.515} C_VEL
LIN {X 0,Y 346.142,Z 1149.099,A -85,B 0,C 180,E1 9061.346,E2 9061.346} C_VEL
LIN {X 0,Y 351.885,Z 1138.615,A -85,B 0,C 180,E1 9058.094,E2 9058.094} C_VEL
LIN {X 0,Y 358.172,Z 1127.447,A -85,B 0,C 180,E1 9055.09,E2 9055.09} C_VEL
LIN {X 0,Y 365.664,Z 1114.311,A -85,B 0,C 180,E1 9052.03,E2 9052.03} C_VEL
LIN {X 0,Y 375.787,Z 1096.42,A -85,B 0,C 180,E1 9048.506,E2 9048.506} C_VEL
LIN {X 0,Y 384.413,Z 1080.641,A -85,B 0,C 180,E1 9045.89,E2 9045.89} C_VEL
LIN {X 0,Y 386.351,Z 1075.815,A -85,B 0,C 180,E1 9045.042,E2 9045.042} C_VEL
LIN {X 0,Y 388.952,Z 1063.209,A -85,B 0,C 180,E1 9042.542,E2 9042.542} C_VEL
LIN {X 0,Y 390.877,Z 1058.762,A -85,B 0,C 180,E1 9041.865,E2 9041.865} C_VEL
LIN {X 0,Y 401.417,Z 1037.938,A -85,B 0,C 180,E1 9039.45,E2 9039.45} C_VEL
LIN {X 0,Y 409.91,Z 1020.146,A -85,B 0,C 180,E1 9037.689,E2 9037.689} C_VEL
LIN {X 0,Y 417.602,Z 1002.94,A -85,B 0,C 180,E1 9036.206,E2 9036.206} C_VEL
LIN {X 0,Y 425.14,Z 984.746,A -85,B 0,C 180,E1 9034.834,E2 9034.834} C_VEL
LIN {X 0,Y 433.915,Z 961.738,A -85,B 0,C 180,E1 9033.351,E2 9033.351} C_VEL
LIN {X 0,Y 442.251,Z 936.702,A -85,B 0,C 180,E1 9032.023,E2 9032.023} C_VEL
LIN {X 0,Y 448.396,Z 915.819,A -85,B 0,C 180,E1 9031.098,E2 9031.098} C_VEL
LIN {X 0,Y 453.597,Z 895.703,A -85,B 0,C 180,E1 9030.345,E2 9030.345} C_VEL
LIN {X 0,Y 458.38,Z 874.151,A -85,B 0,C 180,E1 9029.67,E2 9029.67} C_VEL
LIN {X 0,Y 463.338,Z 847.124,A -85,B 0,C 180,E1 9029.003,E2 9029.003} C_VEL
LIN {X 0,Y 466.765,Z 820.115,A -85,B 0,C 180,E1 9028.5,E2 9028.5} C_VEL
LIN {X 0,Y 477.544,Z 684.439,A -85,B 0,C 180,E1 9026.378,E2 9026.378} C_VEL
LIN {X 0,Y 487.839,Z 555.514,A -85,B 0,C 180,E1 9024.375,E2 9024.375} C_VEL
LIN {X 0,Y 481.006,Z 544.224,A -85,B 0,C 180,E1 9021.621,E2 9021.621} C_VEL
LIN {X 0,Y 475.729,Z 535.833,A -85,B 0,C 180,E1 9019.14,E2 9019.14} C_VEL
LIN {X 0,Y 472.017,Z 530.249,A -85,B 0,C 180,E1 9017.125,E2 9017.125} C_VEL
LIN {X 0,Y 469.701,Z 526.696,A -85,B 0,C 180,E1 9015.686,E2 9015.686} C_VEL
LIN {X 0,Y 467.002,Z 522.541,A -85,B 0,C 180,E1 9013.749,E2 9013.749} C_VEL
LIN {X 0,Y 463.908,Z 517.757,A -85,B 0,C 180,E1 9010.934,E2 9010.934} C_VEL
LIN {X 0,Y 461.505,Z 514.432,A -85,B 0,C 180,E1 9007.72,E2 9007.72} C_VEL
LIN {X 0,Y 460.913,Z 512.632,A -85,B 0,C 180,E1 9006.227,E2 9006.227} C_VEL
LIN {X 0,Y 460.764,Z 512.594,A -85,B 0,C 180,E1 9000.249,E2 9000.249} C_VEL
LIN {X 0,Y 461.095,Z 513.079,A -85,B 0,C 180,E1 8999.379,E2 8999.379} C_VEL
LIN {X 0,Y 462.886,Z 516.816,A -85,B 0,C 180,E1 8996.284,E2 8996.284} C_VEL
LIN {X 0,Y 464.423,Z 518.618,A -85,B 0,C 180,E1 8994.626,E2 8994.626} C_VEL
LIN {X 0,Y 468.014,Z 524.156,A -85,B 0,C 180,E1 8991.585,E2 8991.585} C_VEL
LIN {X 0,Y 470.981,Z 528.644,A -85,B 0,C 180,E1 8989.604,E2 8989.604} C_VEL
LIN {X 0,Y 475.296,Z 535.312,A -85,B 0,C 180,E1 8987.177,E2 8987.177} C_VEL
LIN {X 0,Y 480.415,Z 543.437,A -85,B 0,C 180,E1 8984.735,E2 8984.735} C_VEL
LIN {X 0,Y 486.224,Z 552.823,A -85,B 0,C 180,E1 8982.343,E2 8982.343} C_VEL
LIN {X 0,Y 487.913,Z 556.241,A -85,B 0,C 180,E1 8981.678,E2 8981.678} C_VEL
LIN {X 0,Y 470.406,Z 777.371,A -85,B 0,C 180,E1 8978.255,E2 8978.255} C_VEL
LIN {X 0,Y 466.169,Z 828.393,A -85,B 0,C 180,E1 8977.44,E2 8977.44} C_VEL
LIN {X 0,Y 462.047,Z 857.55,A -85,B 0,C 180,E1 8976.869,E2 8976.869} C_VEL
LIN {X 0,Y 457.804,Z 879.967,A -85,B 0,C 180,E1 8976.309,E2 8976.309} C_VEL
LIN {X 0,Y 453.181,Z 900.484,A -85,B 0,C 180,E1 8975.676,E2 8975.676} C_VEL
LIN {X 0,Y 447.644,Z 921.69,A -85,B 0,C 180,E1 8974.887,E2 8974.887} C_VEL
LIN {X 0,Y 440.256,Z 946.46,A -85,B 0,C 180,E1 8973.779,E2 8973.779} C_VEL
LIN {X 0,Y 431.901,Z 970.502,A -85,B 0,C 180,E1 8972.458,E2 8972.458} C_VEL
LIN {X 0,Y 424.263,Z 990.427,A -85,B 0,C 180,E1 8971.164,E2 8971.164} C_VEL
LIN {X 0,Y 416.915,Z 1008.12,A -85,B 0,C 180,E1 8969.835,E2 8969.835} C_VEL
LIN {X 0,Y 408.774,Z 1026.311,A -85,B 0,C 180,E1 8968.271,E2 8968.271} C_VEL
LIN {X 0,Y 398.608,Z 1047.649,A -85,B 0,C 180,E1 8966.129,E2 8966.129} C_VEL
LIN {X 0,Y 387.972,Z 1068.193,A -85,B 0,C 180,E1 8963.647,E2 8963.647} C_VEL
LIN {X 0,Y 379.341,Z 1084.137,A -85,B 0,C 180,E1 8961.401,E2 8961.401} C_VEL
LIN {X 0,Y 371.027,Z 1099.005,A -85,B 0,C 180,E1 8958.988,E2 8958.988} C_VEL
LIN {X 0,Y 361.372,Z 1116.004,A -85,B 0,C 180,E1 8955.777,E2 8955.777} C_VEL
LIN {X 0,Y 352.058,Z 1131.905,A -85,B 0,C 180,E1 8952.16,E2 8952.16} C_VEL
LIN {X 0,Y 345.09,Z 1143.914,A -85,B 0,C 180,E1 8948.958,E2 8948.958} C_VEL
LIN {X 0,Y 339.158,Z 1154.435,A -85,B 0,C 180,E1 8945.714,E2 8945.714} C_VEL
LIN {X 0,Y 333.413,Z 1165.171,A -85,B 0,C 180,E1 8941.858,E2 8941.858} C_VEL
LIN {X 0,Y 327.924,Z 1176.261,A -85,B 0,C 180,E1 8937.022,E2 8937.022} C_VEL
LIN {X 0,Y 324.668,Z 1183.762,A -85,B 0,C 180,E1 8933.025,E2 8933.025} C_VEL
LIN {X 0,Y 322.561,Z 1189.479,A -85,B 0,C 180,E1 8929.371,E2 8929.371} C_VEL
LIN {X 0,Y 321.192,Z 1194.176,A -85,B 0,C 180,E1 8925.714,E2 8925.714} C_VEL
LIN {X 0,Y 320.384,Z 1197.883,A -85,B 0,C 180,E1 8922.07,E2 8922.07} C_VEL
LIN {X 0,Y 320.049,Z 1200.511,A -85,B 0,C 180,E1 8918.625,E2 8918.625} C_VEL
LIN {X 0,Y 319.932,Z 1202.29,A -85,B 0,C 180,E1 8915.201,E2 8915.201} C_VEL
LIN {X 0,Y 319.914,Z 1203.233,A -85,B 0,C 180,E1 8911.792,E2 8911.792} C_VEL
LIN {X 0,Y 319.914,Z 1203.348,A -85,B 0,C 180,E1 8908.389,E2 8908.389} C_VEL
LIN {X 0,Y 319.93,Z 1202.573,A -85,B 0,C 180,E1 8904.801,E2 8904.801} C_VEL
LIN {X 0,Y 320.063,Z 1200.886,A -85,B 0,C 180,E1 8901.196,E2 8901.196} C_VEL
LIN {X 0,Y 320.49,Z 1198.125,A -85,B 0,C 180,E1 8897.386,E2 8897.386} C_VEL
LIN {X 0,Y 321.457,Z 1194.347,A -85,B 0,C 180,E1 8893.558,E2 8893.558} C_VEL
LIN {X 0,Y 323.13,Z 1189.433,A -85,B 0,C 180,E1 8889.653,E2 8889.653} C_VEL
LIN {X 0,Y 325.589,Z 1183.642,A -85,B 0,C 180,E1 8885.894,E2 8885.894} C_VEL
LIN {X 0,Y 329.401,Z 1175.949,A -85,B 0,C 180,E1 8881.737,E2 8881.737} C_VEL
LIN {X 0,Y 335.713,Z 1164.648,A -85,B 0,C 180,E1 8876.77,E2 8876.77} C_VEL
LIN {X 0,Y 342.046,Z 1154.169,A -85,B 0,C 180,E1 8872.974,E2 8872.974} C_VEL
LIN {X 0,Y 348.864,Z 1143.374,A -85,B 0,C 180,E1 8869.63,E2 8869.63} C_VEL
LIN {X 0,Y 356.955,Z 1130.789,A -85,B 0,C 180,E1 8866.278,E2 8866.278} C_VEL
LIN {X 0,Y 368.226,Z 1113.267,A -85,B 0,C 180,E1 8862.39,E2 8862.39} C_VEL
LIN {X 0,Y 377.674,Z 1098.274,A -85,B 0,C 180,E1 8859.61,E2 8859.61} C_VEL
LIN {X 0,Y 386.928,Z 1083.219,A -85,B 0,C 180,E1 8857.207,E2 8857.207} C_VEL
LIN {X 0,Y 397.149,Z 1065.979,A -85,B 0,C 180,E1 8854.841,E2 8854.841} C_VEL
LIN {X 0,Y 409.383,Z 1044.022,A -85,B 0,C 180,E1 8852.322,E2 8852.322} C_VEL
LIN {X 0,Y 419.033,Z 1025.417,A -85,B 0,C 180,E1 8850.527,E2 8850.527} C_VEL
LIN {X 0,Y 427.727,Z 1007.521,A -85,B 0,C 180,E1 8849.041,E2 8849.041} C_VEL
LIN {X 0,Y 436.01,Z 989.18,A -85,B 0,C 180,E1 8847.726,E2 8847.726} C_VEL
LIN {X 0,Y 444.842,Z 967.817,A -85,B 0,C 180,E1 8846.406,E2 8846.406} C_VEL
LIN {X 0,Y 454.309,Z 941.91,A -85,B 0,C 180,E1 8845.09,E2 8845.09} C_VEL
LIN {X 0,Y 461.136,Z 920.549,A -85,B 0,C 180,E1 8844.193,E2 8844.193} C_VEL
LIN {X 0,Y 466.894,Z 900.056,A -85,B 0,C 180,E1 8843.474,E2 8843.474} C_VEL
LIN {X 0,Y 472.062,Z 878.706,A -85,B 0,C 180,E1 8842.854,E2 8842.854} C_VEL
LIN {X 0,Y 476.942,Z 854.429,A -85,B 0,C 180,E1 8842.289,E2 8842.289} C_VEL
LIN {X 0,Y 481.123,Z 825.543,A -85,B 0,C 180,E1 8841.763,E2 8841.763} C_VEL
LIN {X 0,Y 487.803,Z 751.295,A -85,B 0,C 180,E1 8840.611,E2 8840.611} C_VEL
LIN {X 0,Y 504.306,Z 565.808,A -85,B 0,C 180,E1 8837.779,E2 8837.779} C_VEL
LIN {X 0,Y 499.89,Z 558.413,A -85,B 0,C 180,E1 8835.309,E2 8835.309} C_VEL
LIN {X 0,Y 497.251,Z 554.088,A -85,B 0,C 180,E1 8833.548,E2 8833.548} C_VEL
LIN {X 0,Y 495.016,Z 550.42,A -85,B 0,C 180,E1 8831.772,E2 8831.772} C_VEL
LIN {X 0,Y 492.378,Z 545.924,A -85,B 0,C 180,E1 8828.996,E2 8828.996} C_VEL
LIN {X 0,Y 490.154,Z 541.689,A -85,B 0,C 180,E1 8823.977,E2 8823.977} C_VEL
LIN {X 0,Y 490.173,Z 540.789,A -85,B 0,C 180,E1 8822.806,E2 8822.806} C_VEL
LIN {X 0,Y 492.432,Z 545.93,A -85,B 0,C 180,E1 8816.741,E2 8816.741} C_VEL
LIN {X 0,Y 495.755,Z 551.607,A -85,B 0,C 180,E1 8813.398,E2 8813.398} C_VEL
LIN {X 0,Y 498.81,Z 556.541,A -85,B 0,C 180,E1 8811.179,E2 8811.179} C_VEL
LIN {X 0,Y 502.375,Z 562.485,A -85,B 0,C 180,E1 8809.043,E2 8809.043} C_VEL
LIN {X 0,Y 504.237,Z 565.844,A -85,B 0,C 180,E1 8808.044,E2 8808.044} C_VEL
LIN {X 0,Y 484.993,Z 782.521,A -85,B 0,C 180,E1 8804.744,E2 8804.744} C_VEL
LIN {X 0,Y 480.723,Z 827.509,A -85,B 0,C 180,E1 8804.036,E2 8804.036} C_VEL
LIN {X 0,Y 476.382,Z 854.856,A -85,B 0,C 180,E1 8803.507,E2 8803.507} C_VEL
LIN {X 0,Y 471.938,Z 876.695,A -85,B 0,C 180,E1 8802.973,E2 8802.973} C_VEL
LIN {X 0,Y 466.92,Z 897.366,A -85,B 0,C 180,E1 8802.349,E2 8802.349} C_VEL
LIN {X 0,Y 460.64,Z 919.592,A -85,B 0,C 180,E1 8801.541,E2 8801.541} C_VEL
LIN {X 0,Y 451.799,Z 946.377,A -85,B 0,C 180,E1 8800.342,E2 8800.342} C_VEL
LIN {X 0,Y 443.85,Z 967.333,A -85,B 0,C 180,E1 8799.208,E2 8799.208} C_VEL
LIN {X 0,Y 435.75,Z 986.736,A -85,B 0,C 180,E1 8797.973,E2 8797.973} C_VEL
LIN {X 0,Y 427.859,Z 1004.142,A -85,B 0,C 180,E1 8796.693,E2 8796.693} C_VEL
LIN {X 0,Y 418.793,Z 1022.666,A -85,B 0,C 180,E1 8795.127,E2 8795.127} C_VEL
LIN {X 0,Y 407.117,Z 1044.837,A -85,B 0,C 180,E1 8792.909,E2 8792.909} C_VEL
LIN {X 0,Y 396.342,Z 1063.675,A -85,B 0,C 180,E1 8790.645,E2 8790.645} C_VEL
LIN {X 0,Y 387.073,Z 1079.147,A -85,B 0,C 180,E1 8788.477,E2 8788.477} C_VEL
LIN {X 0,Y 377.756,Z 1094.13,A -85,B 0,C 180,E1 8786.048,E2 8786.048} C_VEL
LIN {X 0,Y 366.767,Z 1111.407,A -85,B 0,C 180,E1 8782.753,E2 8782.753} C_VEL
LIN {X 0,Y 356.645,Z 1126.746,A -85,B 0,C 180,E1 8779.196,E2 8779.196} C_VEL
LIN {X 0,Y 349.284,Z 1137.973,A -85,B 0,C 180,E1 8776.15,E2 8776.15} C_VEL
LIN {X 0,Y 342.519,Z 1148.45,A -85,B 0,C 180,E1 8772.856,E2 8772.856} C_VEL
LIN {X 0,Y 335.913,Z 1159.158,A -85,B 0,C 180,E1 8768.906,E2 8768.906} C_VEL
LIN {X 0,Y 329.754,Z 1169.789,A -85,B 0,C 180,E1 8764.121,E2 8764.121} C_VEL
LIN {X 0,Y 325.898,Z 1177.253,A -85,B 0,C 180,E1 8760.005,E2 8760.005} C_VEL
LIN {X 0,Y 323.256,Z 1183.175,A -85,B 0,C 180,E1 8756.054,E2 8756.054} C_VEL
LIN {X 0,Y 321.524,Z 1188,A -85,B 0,C 180,E1 8752.068,E2 8752.068} C_VEL
LIN {X 0,Y 320.457,Z 1192.132,A -85,B 0,C 180,E1 8747.616,E2 8747.616} C_VEL
LIN {X 0,Y 320.014,Z 1194.935,A -85,B 0,C 180,E1 8743,E2 8743} C_VEL
LIN {X 0,Y 319.927,Z 1196.182,A -85,B 0,C 180,E1 8738.99,E2 8738.99} C_VEL
LIN {X 0,Y 319.906,Z 1196.364,A -85,B 0,C 180,E1 8735.2,E2 8735.2} C_VEL
LIN {X 0,Y 319.934,Z 1195.627,A -85,B 0,C 180,E1 8731.611,E2 8731.611} C_VEL
LIN {X 0,Y 320.047,Z 1194.001,A -85,B 0,C 180,E1 8728.03,E2 8728.03} C_VEL
LIN {X 0,Y 320.415,Z 1191.327,A -85,B 0,C 180,E1 8724.268,E2 8724.268} C_VEL
LIN {X 0,Y 321.25,Z 1187.658,A -85,B 0,C 180,E1 8720.504,E2 8720.504} C_VEL
LIN {X 0,Y 322.709,Z 1182.972,A -85,B 0,C 180,E1 8716.745,E2 8716.745} C_VEL
LIN {X 0,Y 324.888,Z 1177.243,A -85,B 0,C 180,E1 8712.999,E2 8712.999} C_VEL
LIN {X 0,Y 327.943,Z 1170.429,A -85,B 0,C 180,E1 8709.287,E2 8709.287} C_VEL
LIN {X 0,Y 333.009,Z 1160.496,A -85,B 0,C 180,E1 8704.762,E2 8704.762} C_VEL
LIN {X 0,Y 339.284,Z 1148.957,A -85,B 0,C 180,E1 8700.517,E2 8700.517} C_VEL
LIN {X 0,Y 345.311,Z 1138.442,A -85,B 0,C 180,E1 8697.215,E2 8697.215} C_VEL
LIN {X 0,Y 352.264,Z 1126.625,A -85,B 0,C 180,E1 8694.016,E2 8694.016} C_VEL
LIN {X 0,Y 361.065,Z 1111.853,A -85,B 0,C 180,E1 8690.591,E2 8690.591} C_VEL
LIN {X 0,Y 371.12,Z 1094.463,A -85,B 0,C 180,E1 8687.238,E2 8687.238} C_VEL
LIN {X 0,Y 379.336,Z 1079.927,A -85,B 0,C 180,E1 8684.842,E2 8684.842} C_VEL
LIN {X 0,Y 387.59,Z 1064.825,A -85,B 0,C 180,E1 8682.673,E2 8682.673} C_VEL
LIN {X 0,Y 390.877,Z 1058.762,A -85,B 0,C 180,E1 8681.865,E2 8681.865} C_VEL
LIN {X 0,Y 393.049,Z 1053.558,A -85,B 0,C 180,E1 8681.083,E2 8681.083} C_VEL
LIN {X 0,Y 395.945,Z 1040.624,A -85,B 0,C 180,E1 8678.884,E2 8678.884} C_VEL
LIN {X 0,Y 398.145,Z 1035.02,A -85,B 0,C 180,E1 8678.175,E2 8678.175} C_VEL
LIN {X 0,Y 407.258,Z 1016.202,A -85,B 0,C 180,E1 8676.361,E2 8676.361} C_VEL
LIN {X 0,Y 418.04,Z 991.953,A -85,B 0,C 180,E1 8674.393,E2 8674.393} C_VEL
LIN {X 0,Y 426.586,Z 970.594,A -85,B 0,C 180,E1 8672.952,E2 8672.952} C_VEL
LIN {X 0,Y 433.582,Z 951.31,A -85,B 0,C 180,E1 8671.832,E2 8671.832} C_VEL
LIN {X 0,Y 440.18,Z 931.217,A -85,B 0,C 180,E1 8670.836,E2 8670.836} C_VEL
LIN {X 0,Y 447.551,Z 905.797,A -85,B 0,C 180,E1 8669.778,E2 8669.778} C_VEL
LIN {X 0,Y 453.791,Z 879.4,A -85,B 0,C 180,E1 8668.911,E2 8668.911} C_VEL
LIN {X 0,Y 458.088,Z 857.523,A -85,B 0,C 180,E1 8668.335,E2 8668.335} C_VEL
LIN {X 0,Y 461.594,Z 835.349,A -85,B 0,C 180,E1 8667.872,E2 8667.872} C_VEL
LIN {X 0,Y 464.658,Z 807.544,A -85,B 0,C 180,E1 8667.392,E2 8667.392} C_VEL
LIN {X 0,Y 482.651,Z 584.498,A -85,B 0,C 180,E1 8663.947,E2 8663.947} C_VEL
LIN {X 0,Y 484.59,Z 560.583,A -85,B 0,C 180,E1 8663.565,E2 8663.565} C_VEL
LIN {X 0,Y 477.506,Z 548.77,A -85,B 0,C 180,E1 8660.533,E2 8660.533} C_VEL
LIN {X 0,Y 472.83,Z 541.328,A -85,B 0,C 180,E1 8658.175,E2 8658.175} C_VEL
LIN {X 0,Y 468.451,Z 534.517,A -85,B 0,C 180,E1 8655.538,E2 8655.538} C_VEL
LIN {X 0,Y 465.715,Z 530.261,A -85,B 0,C 180,E1 8653.534,E2 8653.534} C_VEL
LIN {X 0,Y 462.699,Z 525.547,A -85,B 0,C 180,E1 8650.711,E2 8650.711} C_VEL
LIN {X 0,Y 460.35,Z 522.003,A -85,B 0,C 180,E1 8647.363,E2 8647.363} C_VEL
LIN {X 0,Y 459.889,Z 520.556,A -85,B 0,C 180,E1 8646.116,E2 8646.116} C_VEL
LIN {X 0,Y 459.786,Z 520.535,A -85,B 0,C 180,E1 8640.249,E2 8640.249} C_VEL
LIN {X 0,Y 460.062,Z 520.963,A -85,B 0,C 180,E1 8639.502,E2 8639.502} C_VEL
LIN {X 0,Y 461.804,Z 524.689,A -85,B 0,C 180,E1 8636.4,E2 8636.4} C_VEL
LIN {X 0,Y 463.252,Z 526.418,A -85,B 0,C 180,E1 8634.799,E2 8634.799} C_VEL
LIN {X 0,Y 466.69,Z 531.833,A -85,B 0,C 180,E1 8631.809,E2 8631.809} C_VEL
LIN {X 0,Y 469.594,Z 536.337,A -85,B 0,C 180,E1 8629.821,E2 8629.821} C_VEL
LIN {X 0,Y 474.528,Z 543.979,A -85,B 0,C 180,E1 8627.032,E2 8627.032} C_VEL
LIN {X 0,Y 481.057,Z 554.697,A -85,B 0,C 180,E1 8623.983,E2 8623.983} C_VEL
LIN {X 0,Y 484.681,Z 561.074,A -85,B 0,C 180,E1 8622.49,E2 8622.49} C_VEL
LIN {X 0,Y 466.843,Z 781.176,A -85,B 0,C 180,E1 8619.092,E2 8619.092} C_VEL
LIN {X 0,Y 462.716,Z 829.269,A -85,B 0,C 180,E1 8618.324,E2 8618.324} C_VEL
LIN {X 0,Y 458.547,Z 857.856,A -85,B 0,C 180,E1 8617.765,E2 8617.765} C_VEL
LIN {X 0,Y 454.239,Z 880.171,A -85,B 0,C 180,E1 8617.212,E2 8617.212} C_VEL
LIN {X 0,Y 449.389,Z 901.217,A -85,B 0,C 180,E1 8616.565,E2 8616.565} C_VEL
LIN {X 0,Y 443.604,Z 922.83,A -85,B 0,C 180,E1 8615.763,E2 8615.763} C_VEL
LIN {X 0,Y 435.442,Z 949.179,A -85,B 0,C 180,E1 8614.57,E2 8614.57} C_VEL
LIN {X 0,Y 427.209,Z 972.164,A -85,B 0,C 180,E1 8613.296,E2 8613.296} C_VEL
LIN {X 0,Y 419.496,Z 991.735,A -85,B 0,C 180,E1 8612.018,E2 8612.018} C_VEL
LIN {X 0,Y 411.528,Z 1010.358,A -85,B 0,C 180,E1 8610.607,E2 8610.607} C_VEL
LIN {X 0,Y 401.459,Z 1032.175,A -85,B 0,C 180,E1 8608.681,E2 8608.681} C_VEL
LIN {X 0,Y 390.827,Z 1053.139,A -85,B 0,C 180,E1 8606.453,E2 8606.453} C_VEL
LIN {X 0,Y 382.183,Z 1069.294,A -85,B 0,C 180,E1 8604.454,E2 8604.454} C_VEL
LIN {X 0,Y 373.328,Z 1085.134,A -85,B 0,C 180,E1 8602.195,E2 8602.195} C_VEL
LIN {X 0,Y 363.562,Z 1102.071,A -85,B 0,C 180,E1 8599.382,E2 8599.382} C_VEL
LIN {X 0,Y 352.818,Z 1120.043,A -85,B 0,C 180,E1 8595.8,E2 8595.8} C_VEL
LIN {X 0,Y 344.908,Z 1133.103,A -85,B 0,C 180,E1 8592.716,E2 8592.716} C_VEL
LIN {X 0,Y 337.861,Z 1144.801,A -85,B 0,C 180,E1 8589.516,E2 8589.516} C_VEL
LIN {X 0,Y 330.715,Z 1157.093,A -85,B 0,C 180,E1 8585.58,E2 8585.58} C_VEL
LIN {X 0,Y 324.071,Z 1169.025,A -85,B 0,C 180,E1 8580.935,E2 8580.935} C_VEL
LIN {X 0,Y 319.815,Z 1177.434,A -85,B 0,C 180,E1 8576.995,E2 8576.995} C_VEL
LIN {X 0,Y 316.77,Z 1184.195,A -85,B 0,C 180,E1 8573.239,E2 8573.239} C_VEL
LIN {X 0,Y 314.514,Z 1190.09,A -85,B 0,C 180,E1 8569.308,E2 8569.308} C_VEL
LIN {X 0,Y 312.942,Z 1195.498,A -85,B 0,C 180,E1 8564.81,E2 8564.81} C_VEL
LIN {X 0,Y 312.127,Z 1199.811,A -85,B 0,C 180,E1 8559.776,E2 8559.776} C_VEL
LIN {X 0,Y 311.943,Z 1201.975,A -85,B 0,C 180,E1 8555.888,E2 8555.888} C_VEL
LIN {X 0,Y 311.914,Z 1203.093,A -85,B 0,C 180,E1 8552.205,E2 8552.205} C_VEL
LIN {X 0,Y 311.916,Z 1203.29,A -85,B 0,C 180,E1 8548.531,E2 8548.531} C_VEL
LIN {X 0,Y 311.932,Z 1202.504,A -85,B 0,C 180,E1 8544.667,E2 8544.667} C_VEL
LIN {X 0,Y 312.076,Z 1200.831,A -85,B 0,C 180,E1 8540.968,E2 8540.968} C_VEL
LIN {X 0,Y 312.547,Z 1198.083,A -85,B 0,C 180,E1 8537.06,E2 8537.06} C_VEL
LIN {X 0,Y 313.594,Z 1194.319,A -85,B 0,C 180,E1 8533.134,E2 8533.134} C_VEL
LIN {X 0,Y 315.361,Z 1189.517,A -85,B 0,C 180,E1 8529.201,E2 8529.201} C_VEL
LIN {X 0,Y 318.014,Z 1183.647,A -85,B 0,C 180,E1 8525.282,E2 8525.282} C_VEL
LIN {X 0,Y 321.866,Z 1176.324,A -85,B 0,C 180,E1 8521.217,E2 8521.217} C_VEL
LIN {X 0,Y 328.313,Z 1165.417,A -85,B 0,C 180,E1 8516.247,E2 8516.247} C_VEL
LIN {X 0,Y 335.143,Z 1154.64,A -85,B 0,C 180,E1 8512.244,E2 8512.244} C_VEL
LIN {X 0,Y 342.133,Z 1144.047,A -85,B 0,C 180,E1 8508.887,E2 8508.887} C_VEL
LIN {X 0,Y 350.194,Z 1132.018,A -85,B 0,C 180,E1 8505.612,E2 8505.612} C_VEL
LIN {X 0,Y 360.709,Z 1116.476,A -85,B 0,C 180,E1 8502.023,E2 8502.023} C_VEL
LIN {X 0,Y 371.896,Z 1099.318,A -85,B 0,C 180,E1 8498.769,E2 8498.769} C_VEL
LIN {X 0,Y 381.283,Z 1084.567,A -85,B 0,C 180,E1 8496.384,E2 8496.384} C_VEL
LIN {X 0,Y 391.026,Z 1068.662,A -85,B 0,C 180,E1 8494.165,E2 8494.165} C_VEL
LIN {X 0,Y 402.169,Z 1049.601,A -85,B 0,C 180,E1 8491.894,E2 8491.894} C_VEL
LIN {X 0,Y 414.28,Z 1027.124,A -85,B 0,C 180,E1 8489.674,E2 8489.674} C_VEL
LIN {X 0,Y 423.843,Z 1007.963,A -85,B 0,C 180,E1 8488.081,E2 8488.081} C_VEL
LIN {X 0,Y 432.31,Z 989.683,A -85,B 0,C 180,E1 8486.778,E2 8486.778} C_VEL
LIN {X 0,Y 440.967,Z 969.238,A -85,B 0,C 180,E1 8485.52,E2 8485.52} C_VEL
LIN {X 0,Y 450.978,Z 942.639,A -85,B 0,C 180,E1 8484.17,E2 8484.17} C_VEL
LIN {X 0,Y 458.165,Z 920.616,A -85,B 0,C 180,E1 8483.255,E2 8483.255} C_VEL
LIN {X 0,Y 464.128,Z 899.779,A -85,B 0,C 180,E1 8482.535,E2 8482.535} C_VEL
LIN {X 0,Y 469.313,Z 878.713,A -85,B 0,C 180,E1 8481.932,E2 8481.932} C_VEL
LIN {X 0,Y 474.235,Z 854.657,A -85,B 0,C 180,E1 8481.38,E2 8481.38} C_VEL
LIN {X 0,Y 478.529,Z 825.637,A -85,B 0,C 180,E1 8480.856,E2 8480.856} C_VEL
LIN {X 0,Y 485.137,Z 753.989,A -85,B 0,C 180,E1 8479.75,E2 8479.75} C_VEL
LIN {X 0,Y 501.752,Z 571.542,A -85,B 0,C 180,E1 8476.989,E2 8476.989} C_VEL
LIN {X 0,Y 498.004,Z 565.263,A -85,B 0,C 180,E1 8474.773,E2 8474.773} C_VEL
LIN {X 0,Y 495.8,Z 561.554,A -85,B 0,C 180,E1 8473.232,E2 8473.232} C_VEL
LIN {X 0,Y 493.775,Z 558.149,A -85,B 0,C 180,E1 8471.565,E2 8471.565} C_VEL
LIN {X 0,Y 491.311,Z 553.813,A -85,B 0,C 180,E1 8468.898,E2 8468.898} C_VEL
LIN {X 0,Y 489.167,Z 549.573,A -85,B 0,C 180,E1 8463.868,E2 8463.868} C_VEL
LIN {X 0,Y 489.194,Z 548.745,A -85,B 0,C 180,E1 8462.812,E2 8462.812} C_VEL
LIN {X 0,Y 491.619,Z 554.364,A -85,B 0,C 180,E1 8456.502,E2 8456.502} C_VEL
LIN {X 0,Y 494.55,Z 559.416,A -85,B 0,C 180,E1 8453.557,E2 8453.557} C_VEL
LIN {X 0,Y 497.549,Z 564.373,A -85,B 0,C 180,E1 8451.331,E2 8451.331} C_VEL
LIN {X 0,Y 501.577,Z 571.116,A -85,B 0,C 180,E1 8448.909,E2 8448.909} C_VEL
LIN {X 0,Y 501.664,Z 571.577,A -85,B 0,C 180,E1 8448.843,E2 8448.843} C_VEL
LIN {X 0,Y 481.709,Z 791.549,A -85,B 0,C 180,E1 8445.512,E2 8445.512} C_VEL
LIN {X 0,Y 477.804,Z 829.957,A -85,B 0,C 180,E1 8444.902,E2 8444.902} C_VEL
LIN {X 0,Y 473.577,Z 855.694,A -85,B 0,C 180,E1 8444.406,E2 8444.406} C_VEL
LIN {X 0,Y 469.095,Z 877.245,A -85,B 0,C 180,E1 8443.883,E2 8443.883} C_VEL
LIN {X 0,Y 463.865,Z 898.319,A -85,B 0,C 180,E1 8443.252,E2 8443.252} C_VEL
LIN {X 0,Y 456.882,Z 922.4,A -85,B 0,C 180,E1 8442.377,E2 8442.377} C_VEL
LIN {X 0,Y 448.251,Z 947.602,A -85,B 0,C 180,E1 8441.242,E2 8441.242} C_VEL
LIN {X 0,Y 440.171,Z 968.389,A -85,B 0,C 180,E1 8440.121,E2 8440.121} C_VEL
LIN {X 0,Y 431.911,Z 987.693,A -85,B 0,C 180,E1 8438.897,E2 8438.897} C_VEL
LIN {X 0,Y 423.488,Z 1005.761,A -85,B 0,C 180,E1 8437.569,E2 8437.569} C_VEL
LIN {X 0,Y 412.506,Z 1027.57,A -85,B 0,C 180,E1 8435.696,E2 8435.696} C_VEL
LIN {X 0,Y 400.952,Z 1048.35,A -85,B 0,C 180,E1 8433.54,E2 8433.54} C_VEL
LIN {X 0,Y 391.242,Z 1064.802,A -85,B 0,C 180,E1 8431.538,E2 8431.538} C_VEL
LIN {X 0,Y 381.584,Z 1080.41,A -85,B 0,C 180,E1 8429.332,E2 8429.332} C_VEL
LIN {X 0,Y 370.826,Z 1097.15,A -85,B 0,C 180,E1 8426.565,E2 8426.565} C_VEL
LIN {X 0,Y 359.049,Z 1114.712,A -85,B 0,C 180,E1 8423.056,E2 8423.056} C_VEL
LIN {X 0,Y 350.432,Z 1127.331,A -85,B 0,C 180,E1 8420.059,E2 8420.059} C_VEL
LIN {X 0,Y 342.532,Z 1138.883,A -85,B 0,C 180,E1 8416.866,E2 8416.866} C_VEL
LIN {X 0,Y 335.022,Z 1150.031,A -85,B 0,C 180,E1 8413.261,E2 8413.261} C_VEL
LIN {X 0,Y 326.969,Z 1162.497,A -85,B 0,C 180,E1 8408.372,E2 8408.372} C_VEL
LIN {X 0,Y 321.778,Z 1171.121,A -85,B 0,C 180,E1 8404.223,E2 8404.223} C_VEL
LIN {X 0,Y 318.17,Z 1177.792,A -85,B 0,C 180,E1 8400.394,E2 8400.394} C_VEL
LIN {X 0,Y 315.405,Z 1183.641,A -85,B 0,C 180,E1 8396.347,E2 8396.347} C_VEL
LIN {X 0,Y 313.445,Z 1188.859,A -85,B 0,C 180,E1 8391.829,E2 8391.829} C_VEL
LIN {X 0,Y 312.337,Z 1193.06,A -85,B 0,C 180,E1 8386.744,E2 8386.744} C_VEL
LIN {X 0,Y 311.996,Z 1195.257,A -85,B 0,C 180,E1 8382.586,E2 8382.586} C_VEL
LIN {X 0,Y 311.927,Z 1196.302,A -85,B 0,C 180,E1 8378.85,E2 8378.85} C_VEL
LIN {X 0,Y 311.906,Z 1196.441,A -85,B 0,C 180,E1 8375.149,E2 8375.149} C_VEL
LIN {X 0,Y 311.936,Z 1195.684,A -85,B 0,C 180,E1 8371.469,E2 8371.469} C_VEL
LIN {X 0,Y 312.061,Z 1194.038,A -85,B 0,C 180,E1 8367.796,E2 8367.796} C_VEL
LIN {X 0,Y 312.469,Z 1191.343,A -85,B 0,C 180,E1 8363.938,E2 8363.938} C_VEL
LIN {X 0,Y 313.317,Z 1187.857,A -85,B 0,C 180,E1 8360.262,E2 8360.262} C_VEL
LIN {X 0,Y 314.899,Z 1183.08,A -85,B 0,C 180,E1 8356.322,E2 8356.322} C_VEL
LIN {X 0,Y 317.155,Z 1177.492,A -85,B 0,C 180,E1 8352.572,E2 8352.572} C_VEL
LIN {X 0,Y 320.536,Z 1170.359,A -85,B 0,C 180,E1 8348.594,E2 8348.594} C_VEL
LIN {X 0,Y 325.903,Z 1160.386,A -85,B 0,C 180,E1 8343.977,E2 8343.977} C_VEL
LIN {X 0,Y 332.497,Z 1148.811,A -85,B 0,C 180,E1 8339.654,E2 8339.654} C_VEL
LIN {X 0,Y 338.83,Z 1138.268,A -85,B 0,C 180,E1 8336.304,E2 8336.304} C_VEL
LIN {X 0,Y 345.711,Z 1127.038,A -85,B 0,C 180,E1 8333.223,E2 8333.223} C_VEL
LIN {X 0,Y 354.273,Z 1113.15,A -85,B 0,C 180,E1 8329.947,E2 8329.947} C_VEL
LIN {X 0,Y 365.197,Z 1094.975,A -85,B 0,C 180,E1 8326.373,E2 8326.373} C_VEL
LIN {X 0,Y 374.174,Z 1079.571,A -85,B 0,C 180,E1 8323.821,E2 8323.821} C_VEL
LIN {X 0,Y 382.706,Z 1064.424,A -85,B 0,C 180,E1 8321.649,E2 8321.649} C_VEL
LIN {X 0,Y 391.411,Z 1048.229,A -85,B 0,C 180,E1 8319.628,E2 8319.628} C_VEL
LIN {X 0,Y 398.145,Z 1035.02,A -85,B 0,C 180,E1 8318.175,E2 8318.175} C_VEL
LIN {X 0,Y 400.406,Z 1029.442,A -85,B 0,C 180,E1 8317.477,E2 8317.477} C_VEL
LIN {X 0,Y 403.82,Z 1015.66,A -85,B 0,C 180,E1 8315.438,E2 8315.438} C_VEL
LIN {X 0,Y 406.03,Z 1009.69,A -85,B 0,C 180,E1 8314.812,E2 8314.812} C_VEL
LIN {X 0,Y 415.233,Z 988.841,A -85,B 0,C 180,E1 8313.198,E2 8313.198} C_VEL
LIN {X 0,Y 422.984,Z 969.769,A -85,B 0,C 180,E1 8311.937,E2 8311.937} C_VEL
LIN {X 0,Y 430.206,Z 950.205,A -85,B 0,C 180,E1 8310.819,E2 8310.819} C_VEL
LIN {X 0,Y 437.602,Z 927.937,A -85,B 0,C 180,E1 8309.742,E2 8309.742} C_VEL
LIN {X 0,Y 445.239,Z 901.032,A -85,B 0,C 180,E1 8308.678,E2 8308.678} C_VEL
LIN {X 0,Y 450.658,Z 878.174,A -85,B 0,C 180,E1 8307.95,E2 8307.95} C_VEL
LIN {X 0,Y 454.962,Z 856.461,A -85,B 0,C 180,E1 8307.392,E2 8307.392} C_VEL
LIN {X 0,Y 458.69,Z 832.895,A -85,B 0,C 180,E1 8306.912,E2 8306.912} C_VEL
LIN {X 0,Y 462.288,Z 797.185,A -85,B 0,C 180,E1 8306.32,E2 8306.32} C_VEL
LIN {X 0,Y 480.473,Z 577.542,A -85,B 0,C 180,E1 8302.941,E2 8302.941} C_VEL
LIN {X 0,Y 481.42,Z 565.83,A -85,B 0,C 180,E1 8302.745,E2 8302.745} C_VEL
LIN {X 0,Y 475.295,Z 555.282,A -85,B 0,C 180,E1 8299.99,E2 8299.99} C_VEL
LIN {X 0,Y 470.065,Z 546.838,A -85,B 0,C 180,E1 8297.198,E2 8297.198} C_VEL
LIN {X 0,Y 466.844,Z 541.856,A -85,B 0,C 180,E1 8295.147,E2 8295.147} C_VEL
LIN {X 0,Y 464.426,Z 537.971,A -85,B 0,C 180,E1 8293.313,E2 8293.313} C_VEL
LIN {X 0,Y 461.614,Z 533.433,A -85,B 0,C 180,E1 8290.61,E2 8290.61} C_VEL
LIN {X 0,Y 459.312,Z 529.894,A -85,B 0,C 180,E1 8287.254,E2 8287.254} C_VEL
LIN {X 0,Y 458.867,Z 528.482,A -85,B 0,C 180,E1 8286.004,E2 8286.004} C_VEL
LIN {X 0,Y 458.808,Z 528.476,A -85,B 0,C 180,E1 8280.25,E2 8280.25} C_VEL
LIN {X 0,Y 459.069,Z 529.033,A -85,B 0,C 180,E1 8279.501,E2 8279.501} C_VEL
LIN {X 0,Y 460.923,Z 532.8,A -85,B 0,C 180,E1 8276.267,E2 8276.267} C_VEL
LIN {X 0,Y 462.14,Z 534.341,A -85,B 0,C 180,E1 8274.911,E2 8274.911} C_VEL
LIN {X 0,Y 465.451,Z 539.651,A -85,B 0,C 180,E1 8271.973,E2 8271.973} C_VEL
LIN {X 0,Y 468.305,Z 544.192,A -85,B 0,C 180,E1 8269.979,E2 8269.979} C_VEL
LIN {X 0,Y 472.948,Z 551.515,A -85,B 0,C 180,E1 8267.298,E2 8267.298} C_VEL
LIN {X 0,Y 479.629,Z 562.698,A -85,B 0,C 180,E1 8264.12,E2 8264.12} C_VEL
LIN {X 0,Y 481.523,Z 566.216,A -85,B 0,C 180,E1 8263.307,E2 8263.307} C_VEL
LIN {X 0,Y 463.208,Z 787.108,A -85,B 0,C 180,E1 8259.91,E2 8259.91} C_VEL
LIN {X 0,Y 459.216,Z 831.677,A -85,B 0,C 180,E1 8259.196,E2 8259.196} C_VEL
LIN {X 0,Y 454.985,Z 859.106,A -85,B 0,C 180,E1 8258.653,E2 8258.653} C_VEL
LIN {X 0,Y 450.716,Z 880.681,A -85,B 0,C 180,E1 8258.119,E2 8258.119} C_VEL
LIN {X 0,Y 445.714,Z 901.898,A -85,B 0,C 180,E1 8257.471,E2 8257.471} C_VEL
LIN {X 0,Y 439.318,Z 925.2,A -85,B 0,C 180,E1 8256.606,E2 8256.606} C_VEL
LIN {X 0,Y 430.636,Z 952.042,A -85,B 0,C 180,E1 8255.369,E2 8255.369} C_VEL
LIN {X 0,Y 423.055,Z 972.674,A -85,B 0,C 180,E1 8254.222,E2 8254.222} C_VEL
LIN {X 0,Y 415.314,Z 991.873,A -85,B 0,C 180,E1 8252.972,E2 8252.972} C_VEL
LIN {X 0,Y 406.956,Z 1010.932,A -85,B 0,C 180,E1 8251.533,E2 8251.533} C_VEL
LIN {X 0,Y 396.142,Z 1033.645,A -85,B 0,C 180,E1 8249.513,E2 8249.513} C_VEL
LIN {X 0,Y 385.775,Z 1053.513,A -85,B 0,C 180,E1 8247.39,E2 8247.39} C_VEL
LIN {X 0,Y 376.762,Z 1069.87,A -85,B 0,C 180,E1 8245.357,E2 8245.357} C_VEL
LIN {X 0,Y 367.662,Z 1085.658,A -85,B 0,C 180,E1 8243.088,E2 8243.088} C_VEL
LIN {X 0,Y 357.105,Z 1103.405,A -85,B 0,C 180,E1 8240.103,E2 8240.103} C_VEL
LIN {X 0,Y 346.532,Z 1120.396,A -85,B 0,C 180,E1 8236.646,E2 8236.646} C_VEL
LIN {X 0,Y 338.72,Z 1132.825,A -85,B 0,C 180,E1 8233.678,E2 8233.678} C_VEL
LIN {X 0,Y 331.392,Z 1144.511,A -85,B 0,C 180,E1 8230.444,E2 8230.444} C_VEL
LIN {X 0,Y 324.33,Z 1156.041,A -85,B 0,C 180,E1 8226.72,E2 8226.72} C_VEL
LIN {X 0,Y 316.982,Z 1168.638,A -85,B 0,C 180,E1 8221.789,E2 8221.789} C_VEL
LIN {X 0,Y 312.534,Z 1176.933,A -85,B 0,C 180,E1 8217.846,E2 8217.846} C_VEL
LIN {X 0,Y 309.146,Z 1184.008,A -85,B 0,C 180,E1 8213.847,E2 8213.847} C_VEL
LIN {X 0,Y 306.728,Z 1189.92,A -85,B 0,C 180,E1 8209.818,E2 8209.818} C_VEL
LIN {X 0,Y 305.089,Z 1195.135,A -85,B 0,C 180,E1 8205.395,E2 8205.395} C_VEL
LIN {X 0,Y 304.167,Z 1199.573,A -85,B 0,C 180,E1 8200.226,E2 8200.226} C_VEL
LIN {X 0,Y 303.947,Z 1201.867,A -85,B 0,C 180,E1 8196.043,E2 8196.043} C_VEL
LIN {X 0,Y 303.914,Z 1203.022,A -85,B 0,C 180,E1 8192.075,E2 8192.075} C_VEL
LIN {X 0,Y 303.914,Z 1203.186,A -85,B 0,C 180,E1 8188.304,E2 8188.304} C_VEL
LIN {X 0,Y 303.934,Z 1202.436,A -85,B 0,C 180,E1 8184.526,E2 8184.526} C_VEL
LIN {X 0,Y 304.105,Z 1200.661,A -85,B 0,C 180,E1 8180.539,E2 8180.539} C_VEL
LIN {X 0,Y 304.647,Z 1197.881,A -85,B 0,C 180,E1 8176.525,E2 8176.525} C_VEL
LIN {X 0,Y 305.739,Z 1194.293,A -85,B 0,C 180,E1 8172.687,E2 8172.687} C_VEL
LIN {X 0,Y 307.65,Z 1189.506,A -85,B 0,C 180,E1 8168.655,E2 8168.655} C_VEL
LIN {X 0,Y 310.474,Z 1183.654,A -85,B 0,C 180,E1 8164.64,E2 8164.64} C_VEL
LIN {X 0,Y 314.418,Z 1176.599,A -85,B 0,C 180,E1 8160.617,E2 8160.617} C_VEL
LIN {X 0,Y 320.699,Z 1166.583,A -85,B 0,C 180,E1 8155.862,E2 8155.862} C_VEL
LIN {X 0,Y 328.471,Z 1154.846,A -85,B 0,C 180,E1 8151.39,E2 8151.39} C_VEL
LIN {X 0,Y 335.85,Z 1144.154,A -85,B 0,C 180,E1 8147.945,E2 8147.945} C_VEL
LIN {X 0,Y 344.255,Z 1132.149,A -85,B 0,C 180,E1 8144.636,E2 8144.636} C_VEL
LIN {X 0,Y 355.174,Z 1116.635,A -85,B 0,C 180,E1 8141.022,E2 8141.022} C_VEL
LIN {X 0,Y 366.753,Z 1099.529,A -85,B 0,C 180,E1 8137.757,E2 8137.757} C_VEL
LIN {X 0,Y 376.433,Z 1084.808,A -85,B 0,C 180,E1 8135.37,E2 8135.37} C_VEL
LIN {X 0,Y 386.401,Z 1069.029,A -85,B 0,C 180,E1 8133.165,E2 8133.165} C_VEL
LIN {X 0,Y 396.908,Z 1051.556,A -85,B 0,C 180,E1 8131.074,E2 8131.074} C_VEL
LIN {X 0,Y 409.998,Z 1028.114,A -85,B 0,C 180,E1 8128.737,E2 8128.737} C_VEL
LIN {X 0,Y 420.082,Z 1008.412,A -85,B 0,C 180,E1 8127.104,E2 8127.104} C_VEL
LIN {X 0,Y 428.73,Z 990.185,A -85,B 0,C 180,E1 8125.814,E2 8125.814} C_VEL
LIN {X 0,Y 437.188,Z 970.692,A -85,B 0,C 180,E1 8124.619,E2 8124.619} C_VEL
LIN {X 0,Y 446.627,Z 946.687,A -85,B 0,C 180,E1 8123.384,E2 8123.384} C_VEL
LIN {X 0,Y 455.08,Z 921.471,A -85,B 0,C 180,E1 8122.334,E2 8122.334} C_VEL
LIN {X 0,Y 461.05,Z 901.122,A -85,B 0,C 180,E1 8121.635,E2 8121.635} C_VEL
LIN {X 0,Y 466.364,Z 880.105,A -85,B 0,C 180,E1 8121.036,E2 8121.036} C_VEL
LIN {X 0,Y 470.947,Z 858.456,A -85,B 0,C 180,E1 8120.535,E2 8120.535} C_VEL
LIN {X 0,Y 475.499,Z 830.778,A -85,B 0,C 180,E1 8120.021,E2 8120.021} C_VEL
LIN {X 0,Y 479.983,Z 785.389,A -85,B 0,C 180,E1 8119.314,E2 8119.314} C_VEL
LIN {X 0,Y 499.257,Z 577.437,A -85,B 0,C 180,E1 8116.182,E2 8116.182} C_VEL
LIN {X 0,Y 495.3,Z 570.394,A -85,B 0,C 180,E1 8113.603,E2 8113.603} C_VEL
LIN {X 0,Y 492.541,Z 565.877,A -85,B 0,C 180,E1 8111.357,E2 8111.357} C_VEL
LIN {X 0,Y 490.152,Z 561.62,A -85,B 0,C 180,E1 8108.682,E2 8108.682} C_VEL
LIN {X 0,Y 488.184,Z 557.211,A -85,B 0,C 180,E1 8103.523,E2 8103.523} C_VEL
LIN {X 0,Y 488.215,Z 556.713,A -85,B 0,C 180,E1 8102.817,E2 8102.817} C_VEL
LIN {X 0,Y 490.494,Z 562.155,A -85,B 0,C 180,E1 8096.669,E2 8096.669} C_VEL
LIN {X 0,Y 493.286,Z 567.091,A -85,B 0,C 180,E1 8093.774,E2 8093.774} C_VEL
LIN {X 0,Y 496.21,Z 572.052,A -85,B 0,C 180,E1 8091.541,E2 8091.541} C_VEL
LIN {X 0,Y 499.198,Z 577.284,A -85,B 0,C 180,E1 8089.651,E2 8089.651} C_VEL
LIN {X 0,Y 478.855,Z 796.824,A -85,B 0,C 180,E1 8086.347,E2 8086.347} C_VEL
LIN {X 0,Y 474.912,Z 832.768,A -85,B 0,C 180,E1 8085.772,E2 8085.772} C_VEL
LIN {X 0,Y 470.912,Z 856.426,A -85,B 0,C 180,E1 8085.316,E2 8085.316} C_VEL
LIN {X 0,Y 466.369,Z 877.816,A -85,B 0,C 180,E1 8084.803,E2 8084.803} C_VEL
LIN {X 0,Y 460.926,Z 899.276,A -85,B 0,C 180,E1 8084.167,E2 8084.167} C_VEL
LIN {X 0,Y 453.222,Z 925.145,A -85,B 0,C 180,E1 8083.228,E2 8083.228} C_VEL
LIN {X 0,Y 444.835,Z 948.786,A -85,B 0,C 180,E1 8082.159,E2 8082.159} C_VEL
LIN {X 0,Y 436.995,Z 968.523,A -85,B 0,C 180,E1 8081.104,E2 8081.104} C_VEL
LIN {X 0,Y 428.567,Z 987.819,A -85,B 0,C 180,E1 8079.892,E2 8079.892} C_VEL
LIN {X 0,Y 419.953,Z 1005.88,A -85,B 0,C 180,E1 8078.58,E2 8078.58} C_VEL
LIN {X 0,Y 408.357,Z 1028.334,A -85,B 0,C 180,E1 8076.662,E2 8076.662} C_VEL
LIN {X 0,Y 396.525,Z 1049.018,A -85,B 0,C 180,E1 8074.518,E2 8074.518} C_VEL
LIN {X 0,Y 386.563,Z 1065.418,A -85,B 0,C 180,E1 8072.521,E2 8072.521} C_VEL
LIN {X 0,Y 376.476,Z 1081.218,A -85,B 0,C 180,E1 8070.28,E2 8070.28} C_VEL
LIN {X 0,Y 364.664,Z 1099.024,A -85,B 0,C 180,E1 8067.305,E2 8067.305} C_VEL
LIN {X 0,Y 352.983,Z 1115.692,A -85,B 0,C 180,E1 8063.9,E2 8063.9} C_VEL
LIN {X 0,Y 344.1,Z 1128.201,A -85,B 0,C 180,E1 8060.88,E2 8060.88} C_VEL
LIN {X 0,Y 335.803,Z 1139.839,A -85,B 0,C 180,E1 8057.597,E2 8057.597} C_VEL
LIN {X 0,Y 326.738,Z 1152.808,A -85,B 0,C 180,E1 8053.253,E2 8053.253} C_VEL
LIN {X 0,Y 319.365,Z 1163.605,A -85,B 0,C 180,E1 8048.767,E2 8048.767} C_VEL
LIN {X 0,Y 314.386,Z 1171.481,A -85,B 0,C 180,E1 8044.859,E2 8044.859} C_VEL
LIN {X 0,Y 310.458,Z 1178.332,A -85,B 0,C 180,E1 8040.802,E2 8040.802} C_VEL
LIN {X 0,Y 307.345,Z 1184.62,A -85,B 0,C 180,E1 8036.259,E2 8036.259} C_VEL
LIN {X 0,Y 305.173,Z 1190.215,A -85,B 0,C 180,E1 8030.923,E2 8030.923} C_VEL
LIN {X 0,Y 304.321,Z 1193.429,A -85,B 0,C 180,E1 8026.609,E2 8026.609} C_VEL
LIN {X 0,Y 304.005,Z 1195.376,A -85,B 0,C 180,E1 8022.73,E2 8022.73} C_VEL
LIN {X 0,Y 303.928,Z 1196.401,A -85,B 0,C 180,E1 8018.894,E2 8018.894} C_VEL
LIN {X 0,Y 303.906,Z 1196.541,A -85,B 0,C 180,E1 8015.285,E2 8015.285} C_VEL
LIN {X 0,Y 303.936,Z 1195.807,A -85,B 0,C 180,E1 8011.507,E2 8011.507} C_VEL
LIN {X 0,Y 304.066,Z 1194.186,A -85,B 0,C 180,E1 8007.738,E2 8007.738} C_VEL
LIN {X 0,Y 304.497,Z 1191.516,A -85,B 0,C 180,E1 8003.778,E2 8003.778} C_VEL
LIN {X 0,Y 305.449,Z 1187.851,A -85,B 0,C 180,E1 7999.818,E2 7999.818} C_VEL
LIN {X 0,Y 307.111,Z 1183.17,A -85,B 0,C 180,E1 7995.866,E2 7995.866} C_VEL
LIN {X 0,Y 309.588,Z 1177.443,A -85,B 0,C 180,E1 7991.937,E2 7991.937} C_VEL
LIN {X 0,Y 313.175,Z 1170.288,A -85,B 0,C 180,E1 7987.867,E2 7987.867} C_VEL
LIN {X 0,Y 319.111,Z 1159.815,A -85,B 0,C 180,E1 7982.977,E2 7982.977} C_VEL
LIN {X 0,Y 325.794,Z 1148.663,A -85,B 0,C 180,E1 7978.756,E2 7978.756} C_VEL
LIN {X 0,Y 332.442,Z 1138.088,A -85,B 0,C 180,E1 7975.357,E2 7975.357} C_VEL
LIN {X 0,Y 340.034,Z 1126.208,A -85,B 0,C 180,E1 7972.079,E2 7972.079} C_VEL
LIN {X 0,Y 349.882,Z 1110.83,A -85,B 0,C 180,E1 7968.47,E2 7968.47} C_VEL
LIN {X 0,Y 360.343,Z 1093.834,A -85,B 0,C 180,E1 7965.186,E2 7965.186} C_VEL
LIN {X 0,Y 369.136,Z 1079.214,A -85,B 0,C 180,E1 7962.772,E2 7962.772} C_VEL
LIN {X 0,Y 378.504,Z 1063.029,A -85,B 0,C 180,E1 7960.465,E2 7960.465} C_VEL
LIN {X 0,Y 389.604,Z 1042.854,A -85,B 0,C 180,E1 7958.011,E2 7958.011} C_VEL
LIN {X 0,Y 400.211,Z 1021.794,A -85,B 0,C 180,E1 7955.889,E2 7955.889} C_VEL
LIN {X 0,Y 406.03,Z 1009.69,A -85,B 0,C 180,E1 7954.812,E2 7954.812} C_VEL
LIN {X 0,Y 408.215,Z 1003.734,A -85,B 0,C 180,E1 7954.203,E2 7954.203} C_VEL
LIN {X 0,Y 411.694,Z 989.039,A -85,B 0,C 180,E1 7952.344,E2 7952.344} C_VEL
LIN {X 0,Y 413.944,Z 982.704,A -85,B 0,C 180,E1 7951.786,E2 7951.786} C_VEL
LIN {X 0,Y 424.079,Z 957.122,A -85,B 0,C 180,E1 7950.217,E2 7950.217} C_VEL
LIN {X 0,Y 431.846,Z 934.809,A -85,B 0,C 180,E1 7949.093,E2 7949.093} C_VEL
LIN {X 0,Y 438.082,Z 914.629,A -85,B 0,C 180,E1 7948.236,E2 7948.236} C_VEL
LIN {X 0,Y 443.588,Z 894.279,A -85,B 0,C 180,E1 7947.504,E2 7947.504} C_VEL
LIN {X 0,Y 449.456,Z 868.853,A -85,B 0,C 180,E1 7946.758,E2 7946.758} C_VEL
LIN {X 0,Y 454.313,Z 841.376,A -85,B 0,C 180,E1 7946.146,E2 7946.146} C_VEL
LIN {X 0,Y 457.243,Z 818.604,A -85,B 0,C 180,E1 7945.74,E2 7945.74} C_VEL
LIN {X 0,Y 475.338,Z 606.482,A -85,B 0,C 180,E1 7942.475,E2 7942.475} C_VEL
LIN {X 0,Y 478.342,Z 570.978,A -85,B 0,C 180,E1 7941.908,E2 7941.908} C_VEL
LIN {X 0,Y 472.644,Z 561.176,A -85,B 0,C 180,E1 7939.206,E2 7939.206} C_VEL
LIN {X 0,Y 468.077,Z 553.677,A -85,B 0,C 180,E1 7936.633,E2 7936.633} C_VEL
LIN {X 0,Y 465.432,Z 549.433,A -85,B 0,C 180,E1 7934.876,E2 7934.876} C_VEL
LIN {X 0,Y 463.159,Z 545.697,A -85,B 0,C 180,E1 7933.102,E2 7933.102} C_VEL
LIN {X 0,Y 460.415,Z 541.221,A -85,B 0,C 180,E1 7930.385,E2 7930.385} C_VEL
LIN {X 0,Y 458.179,Z 537.46,A -85,B 0,C 180,E1 7926.894,E2 7926.894} C_VEL
LIN {X 0,Y 457.847,Z 536.408,A -85,B 0,C 180,E1 7925.891,E2 7925.891} C_VEL
LIN {X 0,Y 457.877,Z 536.439,A -85,B 0,C 180,E1 7920.125,E2 7920.125} C_VEL
LIN {X 0,Y 460.255,Z 541.141,A -85,B 0,C 180,E1 7915.889,E2 7915.889} C_VEL
LIN {X 0,Y 461.083,Z 542.384,A -85,B 0,C 180,E1 7914.961,E2 7914.961} C_VEL
LIN {X 0,Y 464.139,Z 547.328,A -85,B 0,C 180,E1 7912.2,E2 7912.2} C_VEL
LIN {X 0,Y 466.84,Z 551.719,A -85,B 0,C 180,E1 7910.258,E2 7910.258} C_VEL
LIN {X 0,Y 471.268,Z 558.874,A -85,B 0,C 180,E1 7907.626,E2 7907.626} C_VEL
LIN {X 0,Y 477.608,Z 569.716,A -85,B 0,C 180,E1 7904.519,E2 7904.519} C_VEL
LIN {X 0,Y 478.463,Z 571.337,A -85,B 0,C 180,E1 7904.136,E2 7904.136} C_VEL
LIN {X 0,Y 459.683,Z 792.828,A -85,B 0,C 180,E1 7900.744,E2 7900.744} C_VEL
LIN {X 0,Y 455.923,Z 832.78,A -85,B 0,C 180,E1 7900.1,E2 7900.1} C_VEL
LIN {X 0,Y 451.719,Z 859.359,A -85,B 0,C 180,E1 7899.577,E2 7899.577} C_VEL
LIN {X 0,Y 447.397,Z 880.788,A -85,B 0,C 180,E1 7899.052,E2 7899.052} C_VEL
LIN {X 0,Y 442.347,Z 901.813,A -85,B 0,C 180,E1 7898.418,E2 7898.418} C_VEL
LIN {X 0,Y 435.732,Z 925.461,A -85,B 0,C 180,E1 7897.548,E2 7897.548} C_VEL
LIN {X 0,Y 427.257,Z 951.201,A -85,B 0,C 180,E1 7896.377,E2 7896.377} C_VEL
LIN {X 0,Y 419.516,Z 971.917,A -85,B 0,C 180,E1 7895.242,E2 7895.242} C_VEL
LIN {X 0,Y 411.606,Z 991.184,A -85,B 0,C 180,E1 7894.003,E2 7894.003} C_VEL
LIN {X 0,Y 403.529,Z 1009.232,A -85,B 0,C 180,E1 7892.662,E2 7892.662} C_VEL
LIN {X 0,Y 393.469,Z 1030.048,A -85,B 0,C 180,E1 7890.859,E2 7890.859} C_VEL
LIN {X 0,Y 381.625,Z 1052.449,A -85,B 0,C 180,E1 7888.521,E2 7888.521} C_VEL
LIN {X 0,Y 372.036,Z 1069.408,A -85,B 0,C 180,E1 7886.424,E2 7886.424} C_VEL
LIN {X 0,Y 362.656,Z 1085.228,A -85,B 0,C 180,E1 7884.154,E2 7884.154} C_VEL
LIN {X 0,Y 352.251,Z 1102.146,A -85,B 0,C 180,E1 7881.316,E2 7881.316} C_VEL
LIN {X 0,Y 341.25,Z 1119.338,A -85,B 0,C 180,E1 7877.843,E2 7877.843} C_VEL
LIN {X 0,Y 332.671,Z 1132.474,A -85,B 0,C 180,E1 7874.694,E2 7874.694} C_VEL
LIN {X 0,Y 325.013,Z 1144.221,A -85,B 0,C 180,E1 7871.41,E2 7871.41} C_VEL
LIN {X 0,Y 317.949,Z 1155.213,A -85,B 0,C 180,E1 7867.824,E2 7867.824} C_VEL
LIN {X 0,Y 310.387,Z 1167.583,A -85,B 0,C 180,E1 7862.985,E2 7862.985} C_VEL
LIN {X 0,Y 305.158,Z 1176.725,A -85,B 0,C 180,E1 7858.581,E2 7858.581} C_VEL
LIN {X 0,Y 301.556,Z 1183.819,A -85,B 0,C 180,E1 7854.486,E2 7854.486} C_VEL
LIN {X 0,Y 299.068,Z 1189.49,A -85,B 0,C 180,E1 7850.552,E2 7850.552} C_VEL
LIN {X 0,Y 297.37,Z 1194.349,A -85,B 0,C 180,E1 7846.407,E2 7846.407} C_VEL
LIN {X 0,Y 296.407,Z 1198.122,A -85,B 0,C 180,E1 7842.271,E2 7842.271} C_VEL
LIN {X 0,Y 296.001,Z 1201.184,A -85,B 0,C 180,E1 7837.571,E2 7837.571} C_VEL
LIN {X 0,Y 295.916,Z 1202.836,A -85,B 0,C 180,E1 7832.906,E2 7832.906} C_VEL
LIN {X 0,Y 295.916,Z 1203.152,A -85,B 0,C 180,E1 7828.645,E2 7828.645} C_VEL
LIN {X 0,Y 295.937,Z 1202.369,A -85,B 0,C 180,E1 7824.378,E2 7824.378} C_VEL
LIN {X 0,Y 296.125,Z 1200.607,A -85,B 0,C 180,E1 7820.281,E2 7820.281} C_VEL
LIN {X 0,Y 296.721,Z 1197.842,A -85,B 0,C 180,E1 7816.158,E2 7816.158} C_VEL
LIN {X 0,Y 297.971,Z 1194.06,A -85,B 0,C 180,E1 7812.019,E2 7812.019} C_VEL
LIN {X 0,Y 300.097,Z 1189.214,A -85,B 0,C 180,E1 7807.861,E2 7807.861} C_VEL
LIN {X 0,Y 303.151,Z 1183.359,A -85,B 0,C 180,E1 7803.771,E2 7803.771} C_VEL
LIN {X 0,Y 307.783,Z 1175.67,A -85,B 0,C 180,E1 7799.335,E2 7799.335} C_VEL
LIN {X 0,Y 315.297,Z 1164.379,A -85,B 0,C 180,E1 7794.08,E2 7794.08} C_VEL
LIN {X 0,Y 322.663,Z 1153.911,A -85,B 0,C 180,E1 7790.1,E2 7790.1} C_VEL
LIN {X 0,Y 330.489,Z 1143.126,A -85,B 0,C 180,E1 7786.626,E2 7786.626} C_VEL
LIN {X 0,Y 339.838,Z 1130.394,A -85,B 0,C 180,E1 7783.142,E2 7783.142} C_VEL
LIN {X 0,Y 352.38,Z 1113.05,A -85,B 0,C 180,E1 7779.229,E2 7779.229} C_VEL
LIN {X 0,Y 362.299,Z 1098.907,A -85,B 0,C 180,E1 7776.574,E2 7776.574} C_VEL
LIN {X 0,Y 372.317,Z 1084.14,A -85,B 0,C 180,E1 7774.194,E2 7774.194} C_VEL
LIN {X 0,Y 382.276,Z 1068.806,A -85,B 0,C 180,E1 7772.066,E2 7772.066} C_VEL
LIN {X 0,Y 393.41,Z 1050.778,A -85,B 0,C 180,E1 7769.927,E2 7769.927} C_VEL
LIN {X 0,Y 406.652,Z 1027.564,A -85,B 0,C 180,E1 7767.647,E2 7767.647} C_VEL
LIN {X 0,Y 416.447,Z 1008.861,A -85,B 0,C 180,E1 7766.11,E2 7766.11} C_VEL
LIN {X 0,Y 425.274,Z 990.695,A -85,B 0,C 180,E1 7764.834,E2 7764.834} C_VEL
LIN {X 0,Y 433.519,Z 972.156,A -85,B 0,C 180,E1 7763.704,E2 7763.704} C_VEL
LIN {X 0,Y 441.989,Z 951.201,A -85,B 0,C 180,E1 7762.618,E2 7762.618} C_VEL
LIN {X 0,Y 451.722,Z 923.588,A -85,B 0,C 180,E1 7761.447,E2 7761.447} C_VEL
LIN {X 0,Y 458.48,Z 901.049,A -85,B 0,C 180,E1 7760.679,E2 7760.679} C_VEL
LIN {X 0,Y 463.834,Z 880.239,A -85,B 0,C 180,E1 7760.095,E2 7760.095} C_VEL
LIN {X 0,Y 468.476,Z 858.705,A -85,B 0,C 180,E1 7759.605,E2 7759.605} C_VEL
LIN {X 0,Y 473.084,Z 831.383,A -85,B 0,C 180,E1 7759.103,E2 7759.103} C_VEL
LIN {X 0,Y 477.58,Z 787.084,A -85,B 0,C 180,E1 7758.416,E2 7758.416} C_VEL
LIN {X 0,Y 496.862,Z 583.328,A -85,B 0,C 180,E1 7755.367,E2 7755.367} C_VEL
LIN {X 0,Y 493.385,Z 577.188,A -85,B 0,C 180,E1 7752.941,E2 7752.941} C_VEL
LIN {X 0,Y 491.313,Z 573.604,A -85,B 0,C 180,E1 7751.148,E2 7751.148} C_VEL
LIN {X 0,Y 489.09,Z 569.508,A -85,B 0,C 180,E1 7748.583,E2 7748.583} C_VEL
LIN {X 0,Y 487.205,Z 565.095,A -85,B 0,C 180,E1 7743.412,E2 7743.412} C_VEL
LIN {X 0,Y 487.234,Z 564.686,A -85,B 0,C 180,E1 7742.823,E2 7742.823} C_VEL
LIN {X 0,Y 489.413,Z 570.057,A -85,B 0,C 180,E1 7736.779,E2 7736.779} C_VEL
LIN {X 0,Y 492.154,Z 575.032,A -85,B 0,C 180,E1 7733.877,E2 7733.877} C_VEL
LIN {X 0,Y 494.877,Z 579.731,A -85,B 0,C 180,E1 7731.752,E2 7731.752} C_VEL
LIN {X 0,Y 496.802,Z 583.296,A -85,B 0,C 180,E1 7730.462,E2 7730.462} C_VEL
LIN {X 0,Y 476.072,Z 802.439,A -85,B 0,C 180,E1 7727.187,E2 7727.187} C_VEL
LIN {X 0,Y 472.323,Z 834.383,A -85,B 0,C 180,E1 7726.673,E2 7726.673} C_VEL
LIN {X 0,Y 468.383,Z 857.105,A -85,B 0,C 180,E1 7726.239,E2 7726.239} C_VEL
LIN {X 0,Y 463.772,Z 878.369,A -85,B 0,C 180,E1 7725.734,E2 7725.734} C_VEL
LIN {X 0,Y 458.104,Z 900.251,A -85,B 0,C 180,E1 7725.093,E2 7725.093} C_VEL
LIN {X 0,Y 450.021,Z 926.592,A -85,B 0,C 180,E1 7724.14,E2 7724.14} C_VEL
LIN {X 0,Y 441.536,Z 949.972,A -85,B 0,C 180,E1 7723.089,E2 7723.089} C_VEL
LIN {X 0,Y 433.555,Z 969.592,A -85,B 0,C 180,E1 7722.046,E2 7722.046} C_VEL
LIN {X 0,Y 424.966,Z 988.783,A -85,B 0,C 180,E1 7720.848,E2 7720.848} C_VEL
LIN {X 0,Y 415.377,Z 1008.365,A -85,B 0,C 180,E1 7719.424,E2 7719.424} C_VEL
LIN {X 0,Y 402.602,Z 1032.031,A -85,B 0,C 180,E1 7717.359,E2 7717.359} C_VEL
LIN {X 0,Y 392.217,Z 1049.69,A -85,B 0,C 180,E1 7715.517,E2 7715.517} C_VEL
LIN {X 0,Y 382.003,Z 1066.033,A -85,B 0,C 180,E1 7713.529,E2 7713.529} C_VEL
LIN {X 0,Y 371.64,Z 1081.787,A -85,B 0,C 180,E1 7711.291,E2 7711.291} C_VEL
LIN {X 0,Y 358.922,Z 1100.249,A -85,B 0,C 180,E1 7708.173,E2 7708.173} C_VEL
LIN {X 0,Y 347.791,Z 1115.595,A -85,B 0,C 180,E1 7705.019,E2 7705.019} C_VEL
LIN {X 0,Y 338.662,Z 1127.958,A -85,B 0,C 180,E1 7702.025,E2 7702.025} C_VEL
LIN {X 0,Y 329.98,Z 1139.628,A -85,B 0,C 180,E1 7698.716,E2 7698.716} C_VEL
LIN {X 0,Y 320.665,Z 1152.346,A -85,B 0,C 180,E1 7694.433,E2 7694.433} C_VEL
LIN {X 0,Y 312.642,Z 1163.48,A -85,B 0,C 180,E1 7689.763,E2 7689.763} C_VEL
LIN {X 0,Y 307.166,Z 1171.639,A -85,B 0,C 180,E1 7685.638,E2 7685.638} C_VEL
LIN {X 0,Y 302.934,Z 1178.567,A -85,B 0,C 180,E1 7681.432,E2 7681.432} C_VEL
LIN {X 0,Y 299.391,Z 1185.345,A -85,B 0,C 180,E1 7676.37,E2 7676.37} C_VEL
LIN {X 0,Y 297.221,Z 1190.54,A -85,B 0,C 180,E1 7671.097,E2 7671.097} C_VEL
LIN {X 0,Y 296.357,Z 1193.571,A -85,B 0,C 180,E1 7666.866,E2 7666.866} C_VEL
LIN {X 0,Y 296.013,Z 1195.497,A -85,B 0,C 180,E1 7662.881,E2 7662.881} C_VEL
LIN {X 0,Y 295.93,Z 1196.477,A -85,B 0,C 180,E1 7659.137,E2 7659.137} C_VEL
LIN {X 0,Y 295.907,Z 1196.618,A -85,B 0,C 180,E1 7655.234,E2 7655.234} C_VEL
LIN {X 0,Y 295.938,Z 1195.863,A -85,B 0,C 180,E1 7651.354,E2 7651.354} C_VEL
LIN {X 0,Y 296.085,Z 1194.221,A -85,B 0,C 180,E1 7647.483,E2 7647.483} C_VEL
LIN {X 0,Y 296.564,Z 1191.53,A -85,B 0,C 180,E1 7643.417,E2 7643.417} C_VEL
LIN {X 0,Y 297.532,Z 1188.047,A -85,B 0,C 180,E1 7639.544,E2 7639.544} C_VEL
LIN {X 0,Y 299.287,Z 1183.391,A -85,B 0,C 180,E1 7635.488,E2 7635.488} C_VEL
LIN {X 0,Y 301.899,Z 1177.689,A -85,B 0,C 180,E1 7631.46,E2 7631.46} C_VEL
LIN {X 0,Y 305.668,Z 1170.553,A -85,B 0,C 180,E1 7627.291,E2 7627.291} C_VEL
LIN {X 0,Y 311.621,Z 1160.588,A -85,B 0,C 180,E1 7622.48,E2 7622.48} C_VEL
LIN {X 0,Y 318.855,Z 1149.013,A -85,B 0,C 180,E1 7617.997,E2 7617.997} C_VEL
LIN {X 0,Y 325.775,Z 1138.468,A -85,B 0,C 180,E1 7614.543,E2 7614.543} C_VEL
LIN {X 0,Y 333.227,Z 1127.236,A -85,B 0,C 180,E1 7611.382,E2 7611.382} C_VEL
LIN {X 0,Y 342.433,Z 1113.344,A -85,B 0,C 180,E1 7608.035,E2 7608.035} C_VEL
LIN {X 0,Y 354.119,Z 1095.166,A -85,B 0,C 180,E1 7604.409,E2 7604.409} C_VEL
LIN {X 0,Y 363.682,Z 1079.754,A -85,B 0,C 180,E1 7601.835,E2 7601.835} C_VEL
LIN {X 0,Y 373.018,Z 1064.104,A -85,B 0,C 180,E1 7599.587,E2 7599.587} C_VEL
LIN {X 0,Y 383.163,Z 1046.225,A -85,B 0,C 180,E1 7597.382,E2 7597.382} C_VEL
LIN {X 0,Y 395.068,Z 1023.523,A -85,B 0,C 180,E1 7595.04,E2 7595.04} C_VEL
LIN {X 0,Y 404.226,Z 1004.583,A -85,B 0,C 180,E1 7593.402,E2 7593.402} C_VEL
LIN {X 0,Y 412.287,Z 986.519,A -85,B 0,C 180,E1 7592.047,E2 7592.047} C_VEL
LIN {X 0,Y 413.944,Z 982.704,A -85,B 0,C 180,E1 7591.786,E2 7591.786} C_VEL
LIN {X 0,Y 416.168,Z 976.397,A -85,B 0,C 180,E1 7591.243,E2 7591.243} C_VEL
LIN {X 0,Y 419.612,Z 960.828,A -85,B 0,C 180,E1 7589.555,E2 7589.555} C_VEL
LIN {X 0,Y 421.562,Z 954.23,A -85,B 0,C 180,E1 7589.073,E2 7589.073} C_VEL
LIN {X 0,Y 428.489,Z 934.619,A -85,B 0,C 180,E1 7588.107,E2 7588.107} C_VEL
LIN {X 0,Y 434.77,Z 914.641,A -85,B 0,C 180,E1 7587.268,E2 7587.268} C_VEL
LIN {X 0,Y 440.559,Z 893.577,A -85,B 0,C 180,E1 7586.523,E2 7586.523} C_VEL
LIN {X 0,Y 446.758,Z 866.898,A -85,B 0,C 180,E1 7585.759,E2 7585.759} C_VEL
LIN {X 0,Y 451.403,Z 840.506,A -85,B 0,C 180,E1 7585.189,E2 7585.189} C_VEL
LIN {X 0,Y 454.312,Z 818.018,A -85,B 0,C 180,E1 7584.794,E2 7584.794} C_VEL
LIN {X 0,Y 472.92,Z 604.73,A -85,B 0,C 180,E1 7581.529,E2 7581.529} C_VEL
LIN {X 0,Y 475.385,Z 576.34,A -85,B 0,C 180,E1 7581.08,E2 7581.08} C_VEL
LIN {X 0,Y 469.982,Z 566.786,A -85,B 0,C 180,E1 7578.353,E2 7578.353} C_VEL
LIN {X 0,Y 466.044,Z 560.331,A -85,B 0,C 180,E1 7576.004,E2 7576.004} C_VEL
LIN {X 0,Y 463.783,Z 556.625,A -85,B 0,C 180,E1 7574.419,E2 7574.419} C_VEL
LIN {X 0,Y 461.891,Z 553.415,A -85,B 0,C 180,E1 7572.884,E2 7572.884} C_VEL
LIN {X 0,Y 459.335,Z 549.106,A -85,B 0,C 180,E1 7570.282,E2 7570.282} C_VEL
LIN {X 0,Y 457.149,Z 545.352,A -85,B 0,C 180,E1 7566.783,E2 7566.783} C_VEL
LIN {X 0,Y 456.828,Z 544.335,A -85,B 0,C 180,E1 7565.779,E2 7565.779} C_VEL
LIN {X 0,Y 456.9,Z 544.38,A -85,B 0,C 180,E1 7560.125,E2 7560.125} C_VEL
LIN {X 0,Y 458.872,Z 548.681,A -85,B 0,C 180,E1 7556.358,E2 7556.358} C_VEL
LIN {X 0,Y 459.868,Z 550.061,A -85,B 0,C 180,E1 7555.198,E2 7555.198} C_VEL
LIN {X 0,Y 462.908,Z 555.143,A -85,B 0,C 180,E1 7552.366,E2 7552.366} C_VEL
LIN {X 0,Y 465.474,Z 559.407,A -85,B 0,C 180,E1 7550.479,E2 7550.479} C_VEL
LIN {X 0,Y 469.712,Z 566.406,A -85,B 0,C 180,E1 7547.896,E2 7547.896} C_VEL
LIN {X 0,Y 475.491,Z 576.572,A -85,B 0,C 180,E1 7544.973,E2 7544.973} C_VEL
LIN {X 0,Y 456.253,Z 798.548,A -85,B 0,C 180,E1 7541.59,E2 7541.59} C_VEL
LIN {X 0,Y 452.555,Z 835.031,A -85,B 0,C 180,E1 7540.995,E2 7540.995} C_VEL
LIN {X 0,Y 448.527,Z 859.823,A -85,B 0,C 180,E1 7540.509,E2 7540.509} C_VEL
LIN {X 0,Y 444.143,Z 881.125,A -85,B 0,C 180,E1 7539.992,E2 7539.992} C_VEL
LIN {X 0,Y 438.875,Z 902.601,A -85,B 0,C 180,E1 7539.349,E2 7539.349} C_VEL
LIN {X 0,Y 431.63,Z 927.893,A -85,B 0,C 180,E1 7538.42,E2 7538.42} C_VEL
LIN {X 0,Y 423.252,Z 952.409,A -85,B 0,C 180,E1 7537.296,E2 7537.296} C_VEL
LIN {X 0,Y 415.369,Z 972.989,A -85,B 0,C 180,E1 7536.169,E2 7536.169} C_VEL
LIN {X 0,Y 407.304,Z 992.143,A -85,B 0,C 180,E1 7534.938,E2 7534.938} C_VEL
LIN {X 0,Y 398.359,Z 1011.599,A -85,B 0,C 180,E1 7533.485,E2 7533.485} C_VEL
LIN {X 0,Y 386.275,Z 1035.56,A -85,B 0,C 180,E1 7531.344,E2 7531.344} C_VEL
LIN {X 0,Y 376.333,Z 1053.645,A -85,B 0,C 180,E1 7529.411,E2 7529.411} C_VEL
LIN {X 0,Y 366.827,Z 1069.98,A -85,B 0,C 180,E1 7527.38,E2 7527.38} C_VEL
LIN {X 0,Y 357.197,Z 1085.744,A -85,B 0,C 180,E1 7525.103,E2 7525.103} C_VEL
LIN {X 0,Y 345.417,Z 1104.301,A -85,B 0,C 180,E1 7521.94,E2 7521.94} C_VEL
LIN {X 0,Y 334.646,Z 1120.427,A -85,B 0,C 180,E1 7518.587,E2 7518.587} C_VEL
LIN {X 0,Y 326.26,Z 1132.804,A -85,B 0,C 180,E1 7515.568,E2 7515.568} C_VEL
LIN {X 0,Y 318.326,Z 1144.512,A -85,B 0,C 180,E1 7512.237,E2 7512.237} C_VEL
LIN {X 0,Y 310.145,Z 1156.781,A -85,B 0,C 180,E1 7508.127,E2 7508.127} C_VEL
LIN {X 0,Y 302.55,Z 1168.606,A -85,B 0,C 180,E1 7503.265,E2 7503.265} C_VEL
LIN {X 0,Y 297.588,Z 1176.936,A -85,B 0,C 180,E1 7499.12,E2 7499.12} C_VEL
LIN {X 0,Y 293.999,Z 1183.628,A -85,B 0,C 180,E1 7495.159,E2 7495.159} C_VEL
LIN {X 0,Y 291.341,Z 1189.317,A -85,B 0,C 180,E1 7491.123,E2 7491.123} C_VEL
LIN {X 0,Y 289.507,Z 1194.194,A -85,B 0,C 180,E1 7486.865,E2 7486.865} C_VEL
LIN {X 0,Y 288.46,Z 1197.984,A -85,B 0,C 180,E1 7482.614,E2 7482.614} C_VEL
LIN {X 0,Y 288.011,Z 1200.945,A -85,B 0,C 180,E1 7477.983,E2 7477.983} C_VEL
LIN {X 0,Y 287.917,Z 1202.718,A -85,B 0,C 180,E1 7473.186,E2 7473.186} C_VEL
LIN {X 0,Y 287.916,Z 1203.071,A -85,B 0,C 180,E1 7468.608,E2 7468.608} C_VEL
LIN {X 0,Y 287.94,Z 1202.301,A -85,B 0,C 180,E1 7464.221,E2 7464.221} C_VEL
LIN {X 0,Y 288.15,Z 1200.553,A -85,B 0,C 180,E1 7460.009,E2 7460.009} C_VEL
LIN {X 0,Y 288.806,Z 1197.803,A -85,B 0,C 180,E1 7455.771,E2 7455.771} C_VEL
LIN {X 0,Y 290.157,Z 1194.037,A -85,B 0,C 180,E1 7451.517,E2 7451.517} C_VEL
LIN {X 0,Y 292.426,Z 1189.235,A -85,B 0,C 180,E1 7447.272,E2 7447.272} C_VEL
LIN {X 0,Y 295.714,Z 1183.369,A -85,B 0,C 180,E1 7443.059,E2 7443.059} C_VEL
LIN {X 0,Y 300.379,Z 1176.051,A -85,B 0,C 180,E1 7438.717,E2 7438.717} C_VEL
LIN {X 0,Y 307.913,Z 1165.359,A -85,B 0,C 180,E1 7433.542,E2 7433.542} C_VEL
LIN {X 0,Y 315.888,Z 1154.511,A -85,B 0,C 180,E1 7429.305,E2 7429.305} C_VEL
LIN {X 0,Y 324.298,Z 1143.436,A -85,B 0,C 180,E1 7425.669,E2 7425.669} C_VEL
LIN {X 0,Y 333.684,Z 1131.16,A -85,B 0,C 180,E1 7422.259,E2 7422.259} C_VEL
LIN {X 0,Y 346.08,Z 1114.762,A -85,B 0,C 180,E1 7418.469,E2 7418.469} C_VEL
LIN {X 0,Y 357.412,Z 1099.126,A -85,B 0,C 180,E1 7415.504,E2 7415.504} C_VEL
LIN {X 0,Y 367.732,Z 1084.387,A -85,B 0,C 180,E1 7413.128,E2 7413.128} C_VEL
LIN {X 0,Y 377.97,Z 1069.09,A -85,B 0,C 180,E1 7411.008,E2 7411.008} C_VEL
LIN {X 0,Y 389.04,Z 1051.645,A -85,B 0,C 180,E1 7408.942,E2 7408.942} C_VEL
LIN {X 0,Y 402.743,Z 1028.326,A -85,B 0,C 180,E1 7406.652,E2 7406.652} C_VEL
LIN {X 0,Y 413.29,Z 1008.639,A -85,B 0,C 180,E1 7405.049,E2 7405.049} C_VEL
LIN {X 0,Y 422.323,Z 990.411,A -85,B 0,C 180,E1 7403.787,E2 7403.787} C_VEL
LIN {X 0,Y 430.855,Z 971.574,A -85,B 0,C 180,E1 7402.659,E2 7402.659} C_VEL
LIN {X 0,Y 439.722,Z 949.984,A -85,B 0,C 180,E1 7401.564,E2 7401.564} C_VEL
LIN {X 0,Y 449.322,Z 923.037,A -85,B 0,C 180,E1 7400.449,E2 7400.449} C_VEL
LIN {X 0,Y 455.972,Z 901.227,A -85,B 0,C 180,E1 7399.72,E2 7399.72} C_VEL
LIN {X 0,Y 461.481,Z 880.163,A -85,B 0,C 180,E1 7399.139,E2 7399.139} C_VEL
LIN {X 0,Y 466.219,Z 858.513,A -85,B 0,C 180,E1 7398.656,E2 7398.656} C_VEL
LIN {X 0,Y 470.897,Z 831.123,A -85,B 0,C 180,E1 7398.161,E2 7398.161} C_VEL
LIN {X 0,Y 475.519,Z 786.435,A -85,B 0,C 180,E1 7397.475,E2 7397.475} C_VEL
LIN {X 0,Y 494.573,Z 589.287,A -85,B 0,C 180,E1 7394.549,E2 7394.549} C_VEL
LIN {X 0,Y 491.822,Z 584.415,A -85,B 0,C 180,E1 7392.505,E2 7392.505} C_VEL
LIN {X 0,Y 490.092,Z 581.33,A -85,B 0,C 180,E1 7390.938,E2 7390.938} C_VEL
LIN {X 0,Y 488.029,Z 577.397,A -85,B 0,C 180,E1 7388.483,E2 7388.483} C_VEL
LIN {X 0,Y 486.228,Z 572.978,A -85,B 0,C 180,E1 7383.301,E2 7383.301} C_VEL
LIN {X 0,Y 486.245,Z 572.758,A -85,B 0,C 180,E1 7382.711,E2 7382.711} C_VEL
LIN {X 0,Y 488.334,Z 577.956,A -85,B 0,C 180,E1 7376.89,E2 7376.89} C_VEL
LIN {X 0,Y 490.899,Z 582.706,A -85,B 0,C 180,E1 7374.096,E2 7374.096} C_VEL
LIN {X 0,Y 493.63,Z 587.559,A -85,B 0,C 180,E1 7371.907,E2 7371.907} C_VEL
LIN {X 0,Y 494.5,Z 589.394,A -85,B 0,C 180,E1 7371.279,E2 7371.279} C_VEL
LIN {X 0,Y 473.201,Z 809.912,A -85,B 0,C 180,E1 7368.009,E2 7368.009} C_VEL
LIN {X 0,Y 469.776,Z 836.463,A -85,B 0,C 180,E1 7367.576,E2 7367.576} C_VEL
LIN {X 0,Y 465.869,Z 858.319,A -85,B 0,C 180,E1 7367.16,E2 7367.16} C_VEL
LIN {X 0,Y 461.056,Z 879.948,A -85,B 0,C 180,E1 7366.649,E2 7366.649} C_VEL
LIN {X 0,Y 454.153,Z 905.775,A -85,B 0,C 180,E1 7365.884,E2 7365.884} C_VEL
LIN {X 0,Y 445.91,Z 930.905,A -85,B 0,C 180,E1 7364.946,E2 7364.946} C_VEL
LIN {X 0,Y 438.355,Z 951.162,A -85,B 0,C 180,E1 7364.033,E2 7364.033} C_VEL
LIN {X 0,Y 430.194,Z 970.753,A -85,B 0,C 180,E1 7362.999,E2 7362.999} C_VEL
LIN {X 0,Y 421.092,Z 990.585,A -85,B 0,C 180,E1 7361.765,E2 7361.765} C_VEL
LIN {X 0,Y 409.469,Z 1013.534,A -85,B 0,C 180,E1 7360.071,E2 7360.071} C_VEL
LIN {X 0,Y 398.193,Z 1033.548,A -85,B 0,C 180,E1 7358.29,E2 7358.29} C_VEL
LIN {X 0,Y 388.032,Z 1050.366,A -85,B 0,C 180,E1 7356.538,E2 7356.538} C_VEL
LIN {X 0,Y 377.566,Z 1066.655,A -85,B 0,C 180,E1 7354.559,E2 7354.559} C_VEL
LIN {X 0,Y 366.201,Z 1083.42,A -85,B 0,C 180,E1 7352.166,E2 7352.166} C_VEL
LIN {X 0,Y 352.626,Z 1102.312,A -85,B 0,C 180,E1 7348.905,E2 7348.905} C_VEL
LIN {X 0,Y 342.324,Z 1116.039,A -85,B 0,C 180,E1 7346.048,E2 7346.048} C_VEL
LIN {X 0,Y 332.864,Z 1128.369,A -85,B 0,C 180,E1 7343.036,E2 7343.036} C_VEL
LIN {X 0,Y 323.837,Z 1140.003,A -85,B 0,C 180,E1 7339.696,E2 7339.696} C_VEL
LIN {X 0,Y 313.924,Z 1152.935,A -85,B 0,C 180,E1 7335.256,E2 7335.256} C_VEL
LIN {X 0,Y 305.705,Z 1163.768,A -85,B 0,C 180,E1 7330.606,E2 7330.606} C_VEL
LIN {X 0,Y 299.933,Z 1171.902,A -85,B 0,C 180,E1 7326.397,E2 7326.397} C_VEL
LIN {X 0,Y 295.442,Z 1178.804,A -85,B 0,C 180,E1 7322.095,E2 7322.095} C_VEL
LIN {X 0,Y 291.549,Z 1185.797,A -85,B 0,C 180,E1 7316.696,E2 7316.696} C_VEL
LIN {X 0,Y 289.331,Z 1190.706,A -85,B 0,C 180,E1 7311.488,E2 7311.488} C_VEL
LIN {X 0,Y 288.398,Z 1193.714,A -85,B 0,C 180,E1 7307.138,E2 7307.138} C_VEL
LIN {X 0,Y 288.022,Z 1195.617,A -85,B 0,C 180,E1 7303.04,E2 7303.04} C_VEL
LIN {X 0,Y 287.93,Z 1196.575,A -85,B 0,C 180,E1 7299.191,E2 7299.191} C_VEL
LIN {X 0,Y 287.908,Z 1196.717,A -85,B 0,C 180,E1 7295.38,E2 7295.38} C_VEL
LIN {X 0,Y 287.938,Z 1195.986,A -85,B 0,C 180,E1 7291.392,E2 7291.392} C_VEL
LIN {X 0,Y 288.091,Z 1194.367,A -85,B 0,C 180,E1 7287.413,E2 7287.413} C_VEL
LIN {X 0,Y 288.597,Z 1191.701,A -85,B 0,C 180,E1 7283.234,E2 7283.234} C_VEL
LIN {X 0,Y 289.695,Z 1188.039,A -85,B 0,C 180,E1 7279.056,E2 7279.056} C_VEL
LIN {X 0,Y 291.584,Z 1183.361,A -85,B 0,C 180,E1 7274.893,E2 7274.893} C_VEL
LIN {X 0,Y 294.536,Z 1177.341,A -85,B 0,C 180,E1 7270.567,E2 7270.567} C_VEL
LIN {X 0,Y 299.033,Z 1169.449,A -85,B 0,C 180,E1 7265.924,E2 7265.924} C_VEL
LIN {X 0,Y 305.857,Z 1158.553,A -85,B 0,C 180,E1 7260.793,E2 7260.793} C_VEL
LIN {X 0,Y 312.657,Z 1148.358,A -85,B 0,C 180,E1 7256.848,E2 7256.848} C_VEL
LIN {X 0,Y 319.945,Z 1137.724,A -85,B 0,C 180,E1 7253.351,E2 7253.351} C_VEL
LIN {X 0,Y 328.879,Z 1124.812,A -85,B 0,C 180,E1 7249.74,E2 7249.74} C_VEL
LIN {X 0,Y 340.305,Z 1108.01,A -85,B 0,C 180,E1 7245.864,E2 7245.864} C_VEL
LIN {X 0,Y 350.077,Z 1093.19,A -85,B 0,C 180,E1 7243.014,E2 7243.014} C_VEL
LIN {X 0,Y 359.458,Z 1078.484,A -85,B 0,C 180,E1 7240.589,E2 7240.589} C_VEL
LIN {X 0,Y 369.713,Z 1061.71,A -85,B 0,C 180,E1 7238.219,E2 7238.219} C_VEL
LIN {X 0,Y 382.415,Z 1039.441,A -85,B 0,C 180,E1 7235.594,E2 7235.594} C_VEL
LIN {X 0,Y 392.226,Z 1020.83,A -85,B 0,C 180,E1 7233.762,E2 7233.762} C_VEL
LIN {X 0,Y 401.061,Z 1002.852,A -85,B 0,C 180,E1 7232.244,E2 7232.244} C_VEL
LIN {X 0,Y 409.516,Z 984.186,A -85,B 0,C 180,E1 7230.882,E2 7230.882} C_VEL
LIN {X 0,Y 419.428,Z 960.101,A -85,B 0,C 180,E1 7229.387,E2 7229.387} C_VEL
LIN {X 0,Y 421.562,Z 954.23,A -85,B 0,C 180,E1 7229.073,E2 7229.073} C_VEL
LIN {X 0,Y 423.599,Z 947.572,A -85,B 0,C 180,E1 7228.604,E2 7228.604} C_VEL
LIN {X 0,Y 426.874,Z 931.261,A -85,B 0,C 180,E1 7227.078,E2 7227.078} C_VEL
LIN {X 0,Y 428.665,Z 924.379,A -85,B 0,C 180,E1 7226.666,E2 7226.666} C_VEL
LIN {X 0,Y 435.958,Z 899.317,A -85,B 0,C 180,E1 7225.739,E2 7225.739} C_VEL
LIN {X 0,Y 441.342,Z 877.593,A -85,B 0,C 180,E1 7225.079,E2 7225.079} C_VEL
LIN {X 0,Y 445.843,Z 855.895,A -85,B 0,C 180,E1 7224.548,E2 7224.548} C_VEL
LIN {X 0,Y 450.045,Z 830.217,A -85,B 0,C 180,E1 7224.048,E2 7224.048} C_VEL
LIN {X 0,Y 453.865,Z 792.334,A -85,B 0,C 180,E1 7223.442,E2 7223.442} C_VEL
LIN {X 0,Y 472.543,Z 581.703,A -85,B 0,C 180,E1 7220.247,E2 7220.247} C_VEL
LIN {X 0,Y 467.816,Z 573.296,A -85,B 0,C 180,E1 7217.733,E2 7217.733} C_VEL
LIN {X 0,Y 463.485,Z 565.795,A -85,B 0,C 180,E1 7214.94,E2 7214.94} C_VEL
LIN {X 0,Y 460.489,Z 560.946,A -85,B 0,C 180,E1 7212.541,E2 7212.541} C_VEL
LIN {X 0,Y 458.147,Z 556.891,A -85,B 0,C 180,E1 7210.055,E2 7210.055} C_VEL
LIN {X 0,Y 456.079,Z 553.08,A -85,B 0,C 180,E1 7206.546,E2 7206.546} C_VEL
LIN {X 0,Y 455.811,Z 552.262,A -85,B 0,C 180,E1 7205.665,E2 7205.665} C_VEL
LIN {X 0,Y 455.922,Z 552.326,A -85,B 0,C 180,E1 7200.126,E2 7200.126} C_VEL
LIN {X 0,Y 457.586,Z 556.295,A -85,B 0,C 180,E1 7196.743,E2 7196.743} C_VEL
LIN {X 0,Y 458.712,Z 557.858,A -85,B 0,C 180,E1 7195.374,E2 7195.374} C_VEL
LIN {X 0,Y 461.681,Z 562.958,A -85,B 0,C 180,E1 7192.534,E2 7192.534} C_VEL
LIN {X 0,Y 464.2,Z 567.256,A -85,B 0,C 180,E1 7190.641,E2 7190.641} C_VEL
LIN {X 0,Y 468.216,Z 574.047,A -85,B 0,C 180,E1 7188.139,E2 7188.139} C_VEL
LIN {X 0,Y 472.596,Z 582.088,A -85,B 0,C 180,E1 7185.816,E2 7185.816} C_VEL
LIN {X 0,Y 453.016,Z 803.216,A -85,B 0,C 180,E1 7182.464,E2 7182.464} C_VEL
LIN {X 0,Y 449.299,Z 837.281,A -85,B 0,C 180,E1 7181.904,E2 7181.904} C_VEL
LIN {X 0,Y 445.424,Z 860.448,A -85,B 0,C 180,E1 7181.451,E2 7181.451} C_VEL
LIN {X 0,Y 440.952,Z 881.705,A -85,B 0,C 180,E1 7180.939,E2 7180.939} C_VEL
LIN {X 0,Y 435.466,Z 903.576,A -85,B 0,C 180,E1 7180.289,E2 7180.289} C_VEL
LIN {X 0,Y 427.543,Z 930.268,A -85,B 0,C 180,E1 7179.304,E2 7179.304} C_VEL
LIN {X 0,Y 419.357,Z 953.614,A -85,B 0,C 180,E1 7178.232,E2 7178.232} C_VEL
LIN {X 0,Y 411.712,Z 973.141,A -85,B 0,C 180,E1 7177.169,E2 7177.169} C_VEL
LIN {X 0,Y 403.484,Z 992.27,A -85,B 0,C 180,E1 7175.95,E2 7175.95} C_VEL
LIN {X 0,Y 394.343,Z 1011.703,A -85,B 0,C 180,E1 7174.51,E2 7174.51} C_VEL
LIN {X 0,Y 382.132,Z 1035.366,A -85,B 0,C 180,E1 7172.41,E2 7172.41} C_VEL
LIN {X 0,Y 371.795,Z 1053.707,A -85,B 0,C 180,E1 7170.459,E2 7170.459} C_VEL
LIN {X 0,Y 362.1,Z 1069.93,A -85,B 0,C 180,E1 7168.445,E2 7168.445} C_VEL
LIN {X 0,Y 352.363,Z 1085.435,A -85,B 0,C 180,E1 7166.208,E2 7166.208} C_VEL
LIN {X 0,Y 340.824,Z 1103.071,A -85,B 0,C 180,E1 7163.217,E2 7163.217} C_VEL
LIN {X 0,Y 328.991,Z 1120.237,A -85,B 0,C 180,E1 7159.657,E2 7159.657} C_VEL
LIN {X 0,Y 319.928,Z 1133.133,A -85,B 0,C 180,E1 7156.476,E2 7156.476} C_VEL
LIN {X 0,Y 311.3,Z 1145.387,A -85,B 0,C 180,E1 7152.917,E2 7152.917} C_VEL
LIN {X 0,Y 302.005,Z 1158.774,A -85,B 0,C 180,E1 7148.252,E2 7148.252} C_VEL
LIN {X 0,Y 295.009,Z 1169.191,A -85,B 0,C 180,E1 7143.77,E2 7143.77} C_VEL
LIN {X 0,Y 289.902,Z 1177.386,A -85,B 0,C 180,E1 7139.552,E2 7139.552} C_VEL
LIN {X 0,Y 285.991,Z 1184.364,A -85,B 0,C 180,E1 7135.249,E2 7135.249} C_VEL
LIN {X 0,Y 282.862,Z 1190.959,A -85,B 0,C 180,E1 7130.269,E2 7130.269} C_VEL
LIN {X 0,Y 280.867,Z 1196.54,A -85,B 0,C 180,E1 7124.641,E2 7124.641} C_VEL
LIN {X 0,Y 280.149,Z 1199.781,A -85,B 0,C 180,E1 7120.073,E2 7120.073} C_VEL
LIN {X 0,Y 279.95,Z 1201.679,A -85,B 0,C 180,E1 7116.152,E2 7116.152} C_VEL
LIN {X 0,Y 279.915,Z 1202.761,A -85,B 0,C 180,E1 7112.048,E2 7112.048} C_VEL
LIN {X 0,Y 279.913,Z 1202.92,A -85,B 0,C 180,E1 7107.954,E2 7107.954} C_VEL
LIN {X 0,Y 279.948,Z 1202.165,A -85,B 0,C 180,E1 7103.85,E2 7103.85} C_VEL
LIN {X 0,Y 280.198,Z 1200.386,A -85,B 0,C 180,E1 7099.515,E2 7099.515} C_VEL
LIN {X 0,Y 280.953,Z 1197.604,A -85,B 0,C 180,E1 7095.154,E2 7095.154} C_VEL
LIN {X 0,Y 282.461,Z 1193.807,A -85,B 0,C 180,E1 7090.78,E2 7090.78} C_VEL
LIN {X 0,Y 284.944,Z 1188.975,A -85,B 0,C 180,E1 7086.421,E2 7086.421} C_VEL
LIN {X 0,Y 288.713,Z 1182.774,A -85,B 0,C 180,E1 7081.902,E2 7081.902} C_VEL
LIN {X 0,Y 295.128,Z 1173.583,A -85,B 0,C 180,E1 7076.481,E2 7076.481} C_VEL
LIN {X 0,Y 302.89,Z 1163.149,A -85,B 0,C 180,E1 7071.64,E2 7071.64} C_VEL
LIN {X 0,Y 310.778,Z 1153.07,A -85,B 0,C 180,E1 7067.747,E2 7067.747} C_VEL
LIN {X 0,Y 319.443,Z 1142.216,A -85,B 0,C 180,E1 7064.212,E2 7064.212} C_VEL
LIN {X 0,Y 331.214,Z 1127.515,A -85,B 0,C 180,E1 7060.204,E2 7060.204} C_VEL
LIN {X 0,Y 343.803,Z 1111.104,A -85,B 0,C 180,E1 7056.599,E2 7056.599} C_VEL
LIN {X 0,Y 354.469,Z 1096.841,A -85,B 0,C 180,E1 7053.974,E2 7053.974} C_VEL
LIN {X 0,Y 365.855,Z 1080.985,A -85,B 0,C 180,E1 7051.496,E2 7051.496} C_VEL
LIN {X 0,Y 379.585,Z 1060.724,A -85,B 0,C 180,E1 7048.856,E2 7048.856} C_VEL
LIN {X 0,Y 391.374,Z 1041.876,A -85,B 0,C 180,E1 7046.835,E2 7046.835} C_VEL
LIN {X 0,Y 401.37,Z 1024.789,A -85,B 0,C 180,E1 7045.274,E2 7045.274} C_VEL
LIN {X 0,Y 411.083,Z 1006.884,A -85,B 0,C 180,E1 7043.861,E2 7043.861} C_VEL
LIN {X 0,Y 421.062,Z 986.937,A -85,B 0,C 180,E1 7042.523,E2 7042.523} C_VEL
LIN {X 0,Y 432.458,Z 961.521,A -85,B 0,C 180,E1 7041.107,E2 7041.107} C_VEL
LIN {X 0,Y 441.268,Z 938.972,A -85,B 0,C 180,E1 7040.081,E2 7040.081} C_VEL
LIN {X 0,Y 448.185,Z 919.019,A -85,B 0,C 180,E1 7039.321,E2 7039.321} C_VEL
LIN {X 0,Y 454.358,Z 898.718,A -85,B 0,C 180,E1 7038.673,E2 7038.673} C_VEL
LIN {X 0,Y 459.981,Z 877.147,A -85,B 0,C 180,E1 7038.103,E2 7038.103} C_VEL
LIN {X 0,Y 465.781,Z 849.903,A -85,B 0,C 180,E1 7037.539,E2 7037.539} C_VEL
LIN {X 0,Y 469.719,Z 823.419,A -85,B 0,C 180,E1 7037.093,E2 7037.093} C_VEL
LIN {X 0,Y 486.21,Z 656.947,A -85,B 0,C 180,E1 7034.627,E2 7034.627} C_VEL
LIN {X 0,Y 492.353,Z 595.426,A -85,B 0,C 180,E1 7033.716,E2 7033.716} C_VEL
LIN {X 0,Y 490.096,Z 591.26,A -85,B 0,C 180,E1 7031.892,E2 7031.892} C_VEL
LIN {X 0,Y 488.877,Z 589.054,A -85,B 0,C 180,E1 7030.727,E2 7030.727} C_VEL
LIN {X 0,Y 486.883,Z 585.2,A -85,B 0,C 180,E1 7028.265,E2 7028.265} C_VEL
LIN {X 0,Y 485.262,Z 580.736,A -85,B 0,C 180,E1 7023.071,E2 7023.071} C_VEL
LIN {X 0,Y 485.242,Z 581.169,A -85,B 0,C 180,E1 7022.244,E2 7022.244} C_VEL
LIN {X 0,Y 487.257,Z 585.855,A -85,B 0,C 180,E1 7017,E2 7017} C_VEL
LIN {X 0,Y 489.712,Z 590.511,A -85,B 0,C 180,E1 7014.258,E2 7014.258} C_VEL
LIN {X 0,Y 492.323,Z 595.265,A -85,B 0,C 180,E1 7012.109,E2 7012.109} C_VEL
LIN {X 0,Y 470.802,Z 813.027,A -85,B 0,C 180,E1 7008.904,E2 7008.904} C_VEL
LIN {X 0,Y 467.562,Z 837.262,A -85,B 0,C 180,E1 7008.51,E2 7008.51} C_VEL
LIN {X 0,Y 463.586,Z 859.014,A -85,B 0,C 180,E1 7008.101,E2 7008.101} C_VEL
LIN {X 0,Y 458.594,Z 880.976,A -85,B 0,C 180,E1 7007.589,E2 7007.589} C_VEL
LIN {X 0,Y 451.299,Z 907.468,A -85,B 0,C 180,E1 7006.808,E2 7006.808} C_VEL
LIN {X 0,Y 443.256,Z 931.472,A -85,B 0,C 180,E1 7005.921,E2 7005.921} C_VEL
LIN {X 0,Y 435.711,Z 951.332,A -85,B 0,C 180,E1 7005.04,E2 7005.04} C_VEL
LIN {X 0,Y 427.855,Z 969.893,A -85,B 0,C 180,E1 7004.079,E2 7004.079} C_VEL
LIN {X 0,Y 419.075,Z 988.766,A -85,B 0,C 180,E1 7002.934,E2 7002.934} C_VEL
LIN {X 0,Y 408.99,Z 1008.52,A -85,B 0,C 180,E1 7001.54,E2 7001.54} C_VEL
LIN {X 0,Y 395.496,Z 1032.42,A -85,B 0,C 180,E1 6999.5,E2 6999.5} C_VEL
LIN {X 0,Y 384.374,Z 1050.418,A -85,B 0,C 180,E1 6997.651,E2 6997.651} C_VEL
LIN {X 0,Y 373.958,Z 1066.241,A -85,B 0,C 180,E1 6995.747,E2 6995.747} C_VEL
LIN {X 0,Y 363.006,Z 1081.984,A -85,B 0,C 180,E1 6993.531,E2 6993.531} C_VEL
LIN {X 0,Y 350.063,Z 1099.69,A -85,B 0,C 180,E1 6990.575,E2 6990.575} C_VEL
LIN {X 0,Y 337.544,Z 1115.773,A -85,B 0,C 180,E1 6987.273,E2 6987.273} C_VEL
LIN {X 0,Y 327.698,Z 1128.131,A -85,B 0,C 180,E1 6984.253,E2 6984.253} C_VEL
LIN {X 0,Y 318.259,Z 1139.797,A -85,B 0,C 180,E1 6980.894,E2 6980.894} C_VEL
LIN {X 0,Y 308.12,Z 1152.448,A -85,B 0,C 180,E1 6976.53,E2 6976.53} C_VEL
LIN {X 0,Y 299.157,Z 1163.647,A -85,B 0,C 180,E1 6971.69,E2 6971.69} C_VEL
LIN {X 0,Y 293.01,Z 1171.807,A -85,B 0,C 180,E1 6967.402,E2 6967.402} C_VEL
LIN {X 0,Y 288.182,Z 1178.735,A -85,B 0,C 180,E1 6963.005,E2 6963.005} C_VEL
LIN {X 0,Y 284.094,Z 1185.514,A -85,B 0,C 180,E1 6957.682,E2 6957.682} C_VEL
LIN {X 0,Y 281.522,Z 1190.713,A -85,B 0,C 180,E1 6952.115,E2 6952.115} C_VEL
LIN {X 0,Y 280.472,Z 1193.745,A -85,B 0,C 180,E1 6947.638,E2 6947.638} C_VEL
LIN {X 0,Y 280.043,Z 1195.671,A -85,B 0,C 180,E1 6943.419,E2 6943.419} C_VEL
LIN {X 0,Y 279.932,Z 1196.652,A -85,B 0,C 180,E1 6939.456,E2 6939.456} C_VEL
LIN {X 0,Y 279.908,Z 1196.817,A -85,B 0,C 180,E1 6935.534,E2 6935.534} C_VEL
LIN {X 0,Y 279.938,Z 1196.108,A -85,B 0,C 180,E1 6931.432,E2 6931.432} C_VEL
LIN {X 0,Y 280.112,Z 1194.401,A -85,B 0,C 180,E1 6927.135,E2 6927.135} C_VEL
LIN {X 0,Y 280.674,Z 1191.713,A -85,B 0,C 180,E1 6922.837,E2 6922.837} C_VEL
LIN {X 0,Y 281.875,Z 1188.031,A -85,B 0,C 180,E1 6918.542,E2 6918.542} C_VEL
LIN {X 0,Y 283.907,Z 1183.331,A -85,B 0,C 180,E1 6914.265,E2 6914.265} C_VEL
LIN {X 0,Y 286.899,Z 1177.584,A -85,B 0,C 180,E1 6910.028,E2 6910.028} C_VEL
LIN {X 0,Y 291.174,Z 1170.406,A -85,B 0,C 180,E1 6905.664,E2 6905.664} C_VEL
LIN {X 0,Y 298.112,Z 1159.888,A -85,B 0,C 180,E1 6900.459,E2 6900.459} C_VEL
LIN {X 0,Y 305.513,Z 1149.206,A -85,B 0,C 180,E1 6896.194,E2 6896.194} C_VEL
LIN {X 0,Y 313.038,Z 1138.658,A -85,B 0,C 180,E1 6892.635,E2 6892.635} C_VEL
LIN {X 0,Y 321.096,Z 1127.425,A -85,B 0,C 180,E1 6889.396,E2 6889.396} C_VEL
LIN {X 0,Y 331.154,Z 1113.317,A -85,B 0,C 180,E1 6885.941,E2 6885.941} C_VEL
LIN {X 0,Y 343.495,Z 1095.342,A -85,B 0,C 180,E1 6882.322,E2 6882.322} C_VEL
LIN {X 0,Y 353.659,Z 1079.923,A -85,B 0,C 180,E1 6879.735,E2 6879.735} C_VEL
LIN {X 0,Y 363.54,Z 1064.263,A -85,B 0,C 180,E1 6877.487,E2 6877.487} C_VEL
LIN {X 0,Y 374.717,Z 1045.561,A -85,B 0,C 180,E1 6875.196,E2 6875.196} C_VEL
LIN {X 0,Y 387.076,Z 1023.002,A -85,B 0,C 180,E1 6872.909,E2 6872.909} C_VEL
LIN {X 0,Y 396.332,Z 1004.699,A -85,B 0,C 180,E1 6871.352,E2 6871.352} C_VEL
LIN {X 0,Y 404.764,Z 986.615,A -85,B 0,C 180,E1 6870.022,E2 6870.022} C_VEL
LIN {X 0,Y 413.02,Z 967.26,A -85,B 0,C 180,E1 6868.793,E2 6868.793} C_VEL
LIN {X 0,Y 422.44,Z 942.818,A -85,B 0,C 180,E1 6867.488,E2 6867.488} C_VEL
LIN {X 0,Y 428.665,Z 924.379,A -85,B 0,C 180,E1 6866.666,E2 6866.666} C_VEL
LIN {X 0,Y 430.416,Z 917.409,A -85,B 0,C 180,E1 6866.271,E2 6866.271} C_VEL
LIN {X 0,Y 433.265,Z 899.314,A -85,B 0,C 180,E1 6864.848,E2 6864.848} C_VEL
LIN {X 0,Y 434.611,Z 893.203,A -85,B 0,C 180,E1 6864.555,E2 6864.555} C_VEL
LIN {X 0,Y 441.083,Z 865.946,A -85,B 0,C 180,E1 6863.803,E2 6863.803} C_VEL
LIN {X 0,Y 445.713,Z 840.4,A -85,B 0,C 180,E1 6863.271,E2 6863.271} C_VEL
LIN {X 0,Y 448.705,Z 817.963,A -85,B 0,C 180,E1 6862.884,E2 6862.884} C_VEL
LIN {X 0,Y 468.329,Z 602.792,A -85,B 0,C 180,E1 6859.632,E2 6859.632} C_VEL
LIN {X 0,Y 469.76,Z 587.174,A -85,B 0,C 180,E1 6859.393,E2 6859.393} C_VEL
LIN {X 0,Y 465.406,Z 579.316,A -85,B 0,C 180,E1 6856.925,E2 6856.925} C_VEL
LIN {X 0,Y 461.579,Z 572.659,A -85,B 0,C 180,E1 6854.297,E2 6854.297} C_VEL
LIN {X 0,Y 459.376,Z 568.847,A -85,B 0,C 180,E1 6852.444,E2 6852.444} C_VEL
LIN {X 0,Y 457.072,Z 564.777,A -85,B 0,C 180,E1 6849.952,E2 6849.952} C_VEL
LIN {X 0,Y 455.017,Z 560.806,A -85,B 0,C 180,E1 6846.308,E2 6846.308} C_VEL
LIN {X 0,Y 454.795,Z 560.188,A -85,B 0,C 180,E1 6845.551,E2 6845.551} C_VEL
LIN {X 0,Y 454.917,Z 560.283,A -85,B 0,C 180,E1 6840.189,E2 6840.189} C_VEL
LIN {X 0,Y 456.511,Z 564.167,A -85,B 0,C 180,E1 6836.861,E2 6836.861} C_VEL
LIN {X 0,Y 457.609,Z 565.776,A -85,B 0,C 180,E1 6835.488,E2 6835.488} C_VEL
LIN {X 0,Y 460.386,Z 570.633,A -85,B 0,C 180,E1 6832.763,E2 6832.763} C_VEL
LIN {X 0,Y 462.846,Z 574.942,A -85,B 0,C 180,E1 6830.864,E2 6830.864} C_VEL
LIN {X 0,Y 466.728,Z 581.689,A -85,B 0,C 180,E1 6828.382,E2 6828.382} C_VEL
LIN {X 0,Y 469.814,Z 587.48,A -85,B 0,C 180,E1 6826.672,E2 6826.672} C_VEL
LIN {X 0,Y 449.885,Z 807.846,A -85,B 0,C 180,E1 6823.352,E2 6823.352} C_VEL
LIN {X 0,Y 446.386,Z 838.026,A -85,B 0,C 180,E1 6822.852,E2 6822.852} C_VEL
LIN {X 0,Y 442.507,Z 860.737,A -85,B 0,C 180,E1 6822.413,E2 6822.413} C_VEL
LIN {X 0,Y 437.942,Z 882.037,A -85,B 0,C 180,E1 6821.907,E2 6821.907} C_VEL
LIN {X 0,Y 432.135,Z 904.71,A -85,B 0,C 180,E1 6821.239,E2 6821.239} C_VEL
LIN {X 0,Y 423.496,Z 932.775,A -85,B 0,C 180,E1 6820.198,E2 6820.198} C_VEL
LIN {X 0,Y 415.968,Z 953.781,A -85,B 0,C 180,E1 6819.237,E2 6819.237} C_VEL
LIN {X 0,Y 408.181,Z 973.285,A -85,B 0,C 180,E1 6818.187,E2 6818.187} C_VEL
LIN {X 0,Y 399.792,Z 992.395,A -85,B 0,C 180,E1 6816.98,E2 6816.98} C_VEL
LIN {X 0,Y 389.77,Z 1013.221,A -85,B 0,C 180,E1 6815.444,E2 6815.444} C_VEL
LIN {X 0,Y 377.685,Z 1035.937,A -85,B 0,C 180,E1 6813.422,E2 6813.422} C_VEL
LIN {X 0,Y 367.046,Z 1054.332,A -85,B 0,C 180,E1 6811.466,E2 6811.466} C_VEL
LIN {X 0,Y 357.121,Z 1070.49,A -85,B 0,C 180,E1 6809.456,E2 6809.456} C_VEL
LIN {X 0,Y 346.365,Z 1087.11,A -85,B 0,C 180,E1 6807.035,E2 6807.035} C_VEL
LIN {X 0,Y 332.969,Z 1106.7,A -85,B 0,C 180,E1 6803.59,E2 6803.59} C_VEL
LIN {X 0,Y 322.646,Z 1121.161,A -85,B 0,C 180,E1 6800.503,E2 6800.503} C_VEL
LIN {X 0,Y 313.68,Z 1133.457,A -85,B 0,C 180,E1 6797.42,E2 6797.42} C_VEL
LIN {X 0,Y 304.737,Z 1145.674,A -85,B 0,C 180,E1 6793.814,E2 6793.814} C_VEL
LIN {X 0,Y 294.718,Z 1159.457,A -85,B 0,C 180,E1 6788.877,E2 6788.877} C_VEL
LIN {X 0,Y 287.77,Z 1169.371,A -85,B 0,C 180,E1 6784.497,E2 6784.497} C_VEL
LIN {X 0,Y 282.526,Z 1177.36,A -85,B 0,C 180,E1 6780.283,E2 6780.283} C_VEL
LIN {X 0,Y 278.473,Z 1184.17,A -85,B 0,C 180,E1 6775.98,E2 6775.98} C_VEL
LIN {X 0,Y 275.236,Z 1190.525,A -85,B 0,C 180,E1 6771.079,E2 6771.079} C_VEL
LIN {X 0,Y 273.024,Z 1196.236,A -85,B 0,C 180,E1 6765.289,E2 6765.289} C_VEL
LIN {X 0,Y 272.175,Z 1199.656,A -85,B 0,C 180,E1 6760.371,E2 6760.371} C_VEL
LIN {X 0,Y 271.949,Z 1201.639,A -85,B 0,C 180,E1 6756.122,E2 6756.122} C_VEL
LIN {X 0,Y 271.915,Z 1202.666,A -85,B 0,C 180,E1 6752.108,E2 6752.108} C_VEL
LIN {X 0,Y 271.913,Z 1202.84,A -85,B 0,C 180,E1 6747.893,E2 6747.893} C_VEL
LIN {X 0,Y 271.953,Z 1202.099,A -85,B 0,C 180,E1 6743.668,E2 6743.668} C_VEL
LIN {X 0,Y 272.23,Z 1200.333,A -85,B 0,C 180,E1 6739.205,E2 6739.205} C_VEL
LIN {X 0,Y 273.061,Z 1197.566,A -85,B 0,C 180,E1 6734.714,E2 6734.714} C_VEL
LIN {X 0,Y 274.698,Z 1193.786,A -85,B 0,C 180,E1 6730.215,E2 6730.215} C_VEL
LIN {X 0,Y 277.36,Z 1188.969,A -85,B 0,C 180,E1 6725.735,E2 6725.735} C_VEL
LIN {X 0,Y 281.171,Z 1183.091,A -85,B 0,C 180,E1 6721.311,E2 6721.311} C_VEL
LIN {X 0,Y 286.76,Z 1175.409,A -85,B 0,C 180,E1 6716.571,E2 6716.571} C_VEL
LIN {X 0,Y 295.639,Z 1164.133,A -85,B 0,C 180,E1 6711.02,E2 6711.02} C_VEL
LIN {X 0,Y 304.247,Z 1153.624,A -85,B 0,C 180,E1 6706.852,E2 6706.852} C_VEL
LIN {X 0,Y 313.182,Z 1142.901,A -85,B 0,C 180,E1 6703.289,E2 6703.289} C_VEL
LIN {X 0,Y 323.208,Z 1130.811,A -85,B 0,C 180,E1 6699.897,E2 6699.897} C_VEL
LIN {X 0,Y 336.536,Z 1114.385,A -85,B 0,C 180,E1 6696.087,E2 6696.087} C_VEL
LIN {X 0,Y 348.644,Z 1098.735,A -85,B 0,C 180,E1 6693.132,E2 6693.132} C_VEL
LIN {X 0,Y 359.703,Z 1083.858,A -85,B 0,C 180,E1 6690.762,E2 6690.762} C_VEL
LIN {X 0,Y 370.452,Z 1068.664,A -85,B 0,C 180,E1 6688.695,E2 6688.695} C_VEL
LIN {X 0,Y 381.744,Z 1051.748,A -85,B 0,C 180,E1 6686.729,E2 6686.729} C_VEL
LIN {X 0,Y 395.711,Z 1029.146,A -85,B 0,C 180,E1 6684.546,E2 6684.546} C_VEL
LIN {X 0,Y 407.101,Z 1008.797,A -85,B 0,C 180,E1 6682.924,E2 6682.924} C_VEL
